(* POU HTML_DECODE, ST *)
FUNCTION HTML_DECODE : STRING(255)
VAR_INPUT
	IN : STRING(255);
END_VAR
VAR
	pos : INT;
	end : INT;
	tmp : STRING(10);
	code : STRING(1);
END_VAR


(*
version 1.2		17. dec. 2008
programmer 		hugo
tested by		oscat

HTML_DECODE converts HTML coded characters to text. 
&amp; is replaced by & ("Ampersand")
&lt; is replaced by < ("lower than")
&gt; is replaced by > ("greater than")
&quot; is replaced by " ("Quote")
all other &names characters are replaced by their respective character codes.

*)
HTML_DECODE := IN;

(* docode characters encoded by character position *)
pos := FIND(HTML_DECODE, '&');
WHILE pos > 0 DO
	tmp := MID(HTML_DECODE, 2, pos + 1);
	IF tmp = '#x' OR tmp = '#X' THEN
		(* hexadecimal representation found *)
		tmp := MID(HTML_DECODE, 10, pos + 3);
		end := FIND(tmp, ';');
		CODE := CHR_TO_STRING(DWORD_TO_BYTE(HEX_TO_DWORD(LEFT(tmp, end - 1))));
		HTML_DECODE := REPLACE(HTML_DECODE, CODE, end + 3, pos);
	ELSIF LEFT(tmp,1) = '#' THEN
		tmp := MID(HTML_DECODE, 10, pos + 2);
		end := FIND(tmp, ';');
		CODE := CHR_TO_STRING(INT_TO_BYTE(STRING_TO_INT(LEFT(tmp, end - 1))));
		HTML_DECODE := REPLACE(HTML_DECODE, CODE, end + 2, pos);
	ELSE
		(* replace all named characters *)
		tmp := MID(HTML_DECODE, 10, pos + 1);
		end := FIND(tmp, ';');
		CODE := CHR_TO_STRING(CHARCODE(LEFT(tmp, end - 1)));
		HTML_DECODE := REPLACE(HTML_DECODE, CODE, end + 1, pos);
	END_IF;
	(* search for next occurence of encoded characters *)
	pos := FINDP(HTML_DECODE, '&', pos + 1);
END_WHILE;



(* revision history
hm	3. mai. 2008	rev 1.0
	original version

hm	16. jun. 2008	rev 1.1
	changed nested call of replace for better compatibility

hm	17. dec. 2008	rev 1.2
	changed function CHR to CHR_TO_STRING

*)
END_FUNCTION

(* POU HTML_ENCODE, ST *)
FUNCTION HTML_ENCODE : STRING(255)
VAR_INPUT
	IN : STRING(255);
	M : BOOL;
END_VAR
VAR
	pt_in : POINTER TO ARRAY[1..255] OF BYTE;
	pt_out : POINTER TO ARRAY[1..256] OF BYTE;
	pos_in : INT;
	pos_out : INT;
	stop : INT;
	B: BYTE;
	tmp : STRING(10);
	i: INT;
END_VAR


(*
version 1.0		3. mai. 2008
programmer 		hugo
tested by		hugo 

HTML_ENCODE checks a string if it contains reserved HTML characters and converts them to alternative html coding.
& is replaced by &amp; ("Ampersand")
< is replaced by &lt; ("lower than")
> is replaced by &gt; ("greater than")
" is replaced by &quot; ("Quote")

*)
pt_in  := ADR(in);
pt_out := ADR(HTML_ENCODE);

(* scan the input string and convert unallowed characters *)
pos_in := 1;
stop := LEN(in);
FOR pos_out := 1 TO 255 DO
	IF pos_in > stop THEN EXIT; END_IF;
	B := pt_in^[pos_in];
	CASE BYTE_TO_INT(B) OF
		34: (* " detected *)
			IF pos_out > 249 THEN EXIT; END_IF;
			pt_out^[pos_out] := 38;
			pos_out := pos_out + 1;
			pt_out^[pos_out] := 113;
			pos_out := pos_out + 1;
			pt_out^[pos_out] := 117;
			pos_out := pos_out + 1;
			pt_out^[pos_out] := 111;
			pos_out := pos_out + 1;
			pt_out^[pos_out] := 116;
			pos_out := pos_out + 1;
			pt_out^[pos_out] := 59;
		38: (* & detected *)
			IF pos_out > 250 THEN EXIT; END_IF;
			pt_out^[pos_out] := 38;
			pos_out := pos_out + 1;
			pt_out^[pos_out] := 97;
			pos_out := pos_out + 1;
			pt_out^[pos_out] := 109;
			pos_out := pos_out + 1;
			pt_out^[pos_out] := 112;
			pos_out := pos_out + 1;
			pt_out^[pos_out] := 59;
		60: (* < detected *)
			IF pos_out > 251 THEN EXIT; END_IF;
			pt_out^[pos_out] := 38;
			pos_out := pos_out + 1;
			pt_out^[pos_out] := 108;
			pos_out := pos_out + 1;
			pt_out^[pos_out] := 116;
			pos_out := pos_out + 1;
			pt_out^[pos_out] := 59;
		62: (* > detected *)
			IF pos_out > 251 THEN EXIT; END_IF;
			pt_out^[pos_out] := 38;
			pos_out := pos_out + 1;
			pt_out^[pos_out] := 103;
			pos_out := pos_out + 1;
			pt_out^[pos_out] := 116;
			pos_out := pos_out + 1;
			pt_out^[pos_out] := 59;
	ELSE
		IF M AND B > 127 THEN
			tmp := CHARNAME(B);
			(* exit if output string has not enough space *)
			IF pos_out + LEN(tmp) + 2 <= 255 THEN
				pt_out^[pos_out] := 38;
				pos_out := pos_out + 1;
				FOR i := 1 TO LEN(tmp) DO
					pt_out^[pos_out] := CODE(tmp, i);
					pos_out := pos_out + 1;
				END_FOR;
				pt_out^[pos_out] := 59;
			END_IF;
		ELSE
			pt_out^[pos_out] := B;
		END_IF;
	END_CASE
	(* increment in by 1 *)
	pos_in := pos_in + 1;
END_FOR;

(* terminate the output string *)
pt_out^[pos_out] := 0;



(* revision history
hm		3. mai. 2008	rev 1.0
	original version

*)
END_FUNCTION

(* POU HYST, ST *)
FUNCTION_BLOCK HYST
VAR_INPUT
	In : REAL;
	ON : REAL;
	OFF : REAL;
END_VAR
VAR_OUTPUT
	Q : BOOL;
	win : BOOL;
END_VAR
VAR
END_VAR

(*
version 1.0	2. jun. 2008
programmer 	hugo
tested BY	oscat

This Hystereses function has two modes:
1. if on > off then Q will be switched high when in > on and switched low when in < off.
2. if on < off then Q will be switched high when in < on and switched low when in > off.
the output win will be high when in is between low and high.

*)
IF ON >= OFF THEN
	IF IN < OFF THEN
		Q := FALSE;
		WIN := FALSE;
	ELSIF  IN > ON THEN
		Q := TRUE;
		WIN := FALSE;
	ELSE
		WIN := TRUE;
	END_IF;
ELSE
	IF IN > OFF THEN
		Q := FALSE;
		WIN := FALSE;
	ELSIF  IN < ON THEN
		Q := TRUE;
		WIN := FALSE;
	ELSE
		WIN := TRUE;
	END_IF;
END_IF;


(* revision history
hm		2.  jun 2008	rev 1.0
	original version

*)
END_FUNCTION_BLOCK

(* POU HYST_1, ST *)
FUNCTION_BLOCK HYST_1
VAR_INPUT
	In : REAL;
	high : REAL;
	low : REAL;
END_VAR
VAR_OUTPUT
	Q : BOOL;
	win : BOOL;
END_VAR
VAR
END_VAR

(*
version 1.1	2. jun. 2008
programmer 	hugo
tested BY	oscat

this hysteresis function switches the output high if the input signal reaches obove high and will switch to low when the input falls back below low value.
a separate output mid is set if the input stays between low and high value.

*)
IF in < low THEN
	Q := FALSE;
	win := FALSE;
ELSIF in > high THEN
	Q := TRUE;
	win := FALSE;
ELSE
	win := TRUE;
END_IF;

(* code used for rev 1.0
IF Q THEN
	IF in < low THEN q := FALSE; END_IF;
ELSE
	IF in > high THEN q := TRUE; END_IF;
END_IF;
win := in > low AND in < high;
*)


(* revision history
hm		4.  aug. 2006	rev 1.0
	original version

hm		2. jun. 2008	rev 1.1
	improved performance
*)
END_FUNCTION_BLOCK

(* POU HYST_2, ST *)
FUNCTION_BLOCK HYST_2
VAR_INPUT
	IN : REAL;
	VAL : REAL;
	HYS : REAL;
END_VAR
VAR_OUTPUT
	Q : BOOL;
	WIN: BOOL;
END_VAR
VAR
	tmp: REAL;
END_VAR


(*
version 1.2	2. jun. 2008
programmer 	oscat
tested BY	oscat

this hysteresis function switches the output high if the input signal reaches obove val + hys/2 and will switch to low when the input falls back below val - hys/2 value.
a separate output mid is set if the input stays between low and high value.

*)
tmp := val - hys * 0.5;
IF in < tmp THEN
	Q := FALSE;
	win := FALSE;
ELSIF in > tmp + hys THEN
	Q := TRUE;
	win := FALSE;
ELSE
	win := TRUE;
END_IF;

(* code used for 1.2 and before
X := hys * 0.5;
IF Q THEN
	IF in < val - x THEN q := FALSE; END_IF;
ELSE
	IF in > val + x THEN q := TRUE; END_IF;
END_IF;
win := in > val - x AND in < val + x;
*)

(* revision history
hm		4. aug 2006	rev 1.0
	original version

hm		5. jan 2008	rev 1.1
	improved code for better performance

hm		2. jun. 2008	rev 1.2
	improved performance
*)
END_FUNCTION_BLOCK

(* POU HYST_3, ST *)
FUNCTION_BLOCK HYST_3
VAR_INPUT
	in : REAL;
	hyst : REAL;
	val1 : REAL;
	val2 : REAL;
END_VAR
VAR_OUTPUT
	Q1 : BOOL;
	Q2 : BOOL;
END_VAR
VAR
	X: REAL;
END_VAR

(*
version 1.2	5 jan 2008
programmer 	oscat
tested BY	oscat

this is a double hysteresis function. Out1 follows a hysteresis function defined by val1and hyst, while out 2 follows val2 and hyst.
if the input signal is between the two hysteresis switches (val1 and val2) then non of the outputs is active.

*)
X := hyst * 0.5;
IF in < val1 - X THEN
	q1 := TRUE;
ELSIF in > val1 + X THEN
	q1 := FALSE;
END_IF;
IF in < val2 - X THEN
	q2 := FALSE;
ELSIF in > val2 + X THEN
	q2 := TRUE;
END_IF;

(* revision history
hm	22. jan 2007	rev 1.0
	original version

hm	27. dec 2007	rev 1.1
	changed code for better performance

hm	5. jan 2008	rev 1.2
	further performance iprovements

*)
END_FUNCTION_BLOCK

(* POU INC_DEC, ST *)
FUNCTION_BLOCK INC_DEC
VAR_INPUT
	CHa : BOOL;
	CHb : BOOL;
	RST : BOOL;
END_VAR
VAR_OUTPUT
	dir : BOOL;
	cnt : INT;
END_VAR
VAR
	edgea : BOOL;
	clk: BOOL;
	clka: BOOL;
	clkb: BOOL;
	edgeb: BOOL;
	axb: BOOL;
END_VAR

(*
	version 1.0	4 aug 2006
	programmer 	oscat
	tested BY		oscat

incremental decoder with quadruple accuracy.
2 pulses for each channel are created for each directional pulse.
*)
axb := cha XOR chb;

(* create pulses for channel a *)
clka := cha XOR edgea;
edgea := cha;

clkb := chb XOR edgeb;
edgeb := chb;

(* create pulses for both channels *)
clk := clka OR clkb;

(* set the direction output *)
IF axb AND clka THEN dir := TRUE; END_IF;
IF axb AND clkb THEN dir := FALSE; END_IF;

(* increment or decrement the counter *)
IF clk AND dir THEN cnt := cnt + 1; END_IF;
IF clk AND NOT dir THEN cnt := cnt -1; END_IF;

(* reset the counter if rst active *)
IF rst THEN cnt := 0; END_IF;
END_FUNCTION_BLOCK

(* POU INT_TO_BCDC, ST *)
FUNCTION INT_TO_BCDC : BYTE
VAR_INPUT
	IN : INT;
END_VAR
VAR
END_VAR

(*
version 1.1	30. jun. 2008
programmer 	hugo
tested by		tobias

this function converts an integer into a two digit bcd number.
*)
INT_TO_BCDC := SHL(INT_TO_BYTE(IN / INT#10),4) OR INT_TO_BYTE(in MOD INT#10);

(* revision history
hm	13.12.2007
	original version

hm	30.6.2008	rev 1.1
	changed name INT_TO_BCD to INT_TO_BCDC to avoid collision with util.lib
	corrected error in code

*)
END_FUNCTION

(* POU INTERLOCK_4, ST *)
FUNCTION_BLOCK INTERLOCK_4
VAR_INPUT CONSTANT
END_VAR
VAR_INPUT
	I0 : BOOL;
	I1 : BOOL;
	I2 : BOOL;
	I3 : BOOL;
	E : BOOL;
	MODE : INT;

END_VAR
VAR_OUTPUT
	OUT : BYTE;
	TP : BOOL;
END_VAR
VAR
	in: BYTE;
	last: BYTE;
	old: BYTE;
	lmode: INT;
END_VAR

(*
version 1.0	24. oct. 2008
programmer 	hugo
tested by	oscat

INTERLOCK_4 detects one of 4 switches and delivers the number of the switch pressed on the output out
a output tp is true for one cycle if the output has changed.
a setup variable MODE selects between 3 different modes:
MODE = 0, any input active will disable all other inputs
MODE = 1, the input with the highest number will be acepted
mode = 2, the input last pressed will disable all others 

*)
(* check if enable is active *)
IF E THEN
(* reset all vars when there is a mode change on thy fly *)
	IF mode <> lmode THEN
		out := last := old := 0;
		lmode := mode;
	END_IF;
	(* load inputs into in *)
	in.0 := I0;	in.1 := I1;	in.2 := I2;	in.3 := I3;
	(* only execute when there is any change *)
	IF in <> last THEN
		(* only execute when inputs have chages state *)
		CASE mode OF
			0:	(* output directly display inputs as bits in byte out *)
				out := in;

			1:	(* the input with the highest number will be acepted *)
				IF in.3 THEN out := 8;
				ELSIF in.2 THEN out := 4;
				ELSIF in.1 THEN out := 2;
				ELSE out := in;
				END_IF;

			2:	(* input last pressed will be displayed only *)
				last := ((in XOR last) AND in);
				IF last.3 THEN out := 8;
				ELSIF last.2 THEN out := 4;
				ELSIF last.1 THEN out := 2;
				ELSE out := last;
				END_IF;

			3:	(* any input active will disable all other inputs *)
				IF (out AND in) = 0 THEN
					IF in.3 THEN out := 8;
					ELSIF in.2 THEN out := 4;
					ELSIF in.1 THEN out := 2;
					ELSE out := in;
					END_IF;
				END_IF;

		END_CASE;
		last := in;
	END_IF;
	tp := out <> old;
	old := out;
ELSE
	out := last := old := 0;
	lmode := 0;
	tp := FALSE;
END_IF;





(* revision history
hm	24. oct 2008	rev 1.0
	original version

*)
END_FUNCTION_BLOCK

(* POU IP4_CHECK, ST *)
FUNCTION IP4_CHECK : BOOL
VAR_INPUT
	NIP : DWORD;
	LIP : DWORD;
	SM : DWORD;
END_VAR
VAR
END_VAR

(*
version 1.0	4. mar 2008
programmer 	hugo
tested by		oscat

IP4_CHECK testet ob eine Network IP und Local_IP im selben Subnet sind.

*)
IP4_CHECK := (NIP AND sm) = (LIP AND SM);


(* revision history
hm		4. mar 2008	rev 1.0
	original version

*)
END_FUNCTION

(* POU IP4_DECODE, ST *)
FUNCTION IP4_DECODE : DWORD
VAR_INPUT
	str : STRING;
END_VAR
VAR
	d1, d2, d3, d4 : INT;
	s1, s2, s3, s4 : STRING(3);
END_VAR

(*
version 1.0	29. feb 2008
programmer 		kurt
tested by		hugo

IP4_DECODE testet ob ein string eine gültige IPv4 Adresse enthält und gibt die 4 Bytes der IP Adresse als DWORD zurück.

*)
IP4_DECODE := 0;
(* check wheather 3 dots are present *)
IF COUNT_CHAR(str,46) <> 3 THEN RETURN; END_IF;
(* store the positions of the 3 dots *)
d1 := FINDP(str,'.',1);
d2 := FINDP(str,'.',d1+1);
d3 := FINDP(str,'.',d2+1);
IF d1 > 4 OR d2 - d1 > 4 OR d3 - d2 > 4 THEN RETURN; END_IF;
(* store the 3 strings between the dots in d1 .. d4 *)
s1 := LEFT(str,d1-1);
s2 := MID(str,d2-d1-1,d1+1);
s3 := MID(str,d3-d2-1,d2+1);
s4 := RIGHT(str,LEN(str)-d3);
(* check if the 3 strings are numbers only *)
IF NOT IS_NUM(s1) OR NOT IS_NUM(s2) OR NOT IS_NUM(s3) OR NOT IS_NUM(s4) THEN RETURN; END_IF;
(* convert the 4 numbers and check range 0..255 *)
d1 := STRING_TO_INT(s1);
d2 := STRING_TO_INT(s2);
d3 := STRING_TO_INT(s3);
d4 := STRING_TO_INT(s4);
(* check range of numbers *)
IF d1 > 255 OR d2 > 255 OR d3 > 255 OR d4 > 255 THEN RETURN; END_IF;
(* convert to output *)
IP4_DECODE := SHL(INT_TO_DWORD(d1),24) OR SHL(INT_TO_DWORD(d2),16) OR SHL(INT_TO_DWORD(d3),8) OR INT_TO_DWORD(d4);



(* revision history
hm		29. feb 2008	rev 1.0
	original version

*)
END_FUNCTION

(* POU IS_NUM, ST *)
FUNCTION IS_NUM : BOOL
VAR_INPUT
	str : STRING(STRING_LENGTH);
END_VAR
VAR
	L : INT;
	pt : POINTER TO BYTE;
	pos: INT;
END_VAR

(*
version 1.1	29. mar. 2008
programmer 		kurt
tested by		hugo

IS_NUM testet ob in einem string nur Zahlen 0..9 vorkommen.

*)
PT := ADR(str);
L := LEN(str);
FOR pos := 1 TO L DO
	IF NOT (ISC_NUM(pt^)) THEN
		IS_NUM := FALSE;
		RETURN;
	END_IF;
    	PT := PT + 1;
END_FOR;
IS_NUM := L > 0;


(* revision history
hm	29. feb 2008	rev 1.0
	original version

hm	29. mar. 2008	rev 1.1
	changed STRING to STRING(STRING_LENGTH)
*)
END_FUNCTION

(* POU ISC_NUM, ST *)
FUNCTION ISC_NUM : BOOL
VAR_INPUT
	IN : BYTE;
END_VAR
VAR
END_VAR

(*
version 1.0	6. mar 2008
programmer 	oscat
tested by		hugo

ISC_NUM checks if a character is 0..9.

*)
ISC_NUM := IN > 47 AND IN < 58;

(* revision history
hm		6. mar. 2008	rev 1.0
	original version

*)
END_FUNCTION

(* POU IP4_TO_STRING, ST *)
FUNCTION IP4_TO_STRING : STRING(15)
VAR_INPUT
	IP4 : DWORD;
END_VAR
VAR
	tmp : STRING(3);
END_VAR

(*
version 1.0	22. apr. 2008
programmer 	kurt
tested by		hugo

IP4_TO_STRING erzeugt eine IP Adresse als String aus einem DWORD..

*)
IP4_TO_STRING := DWORD_TO_STRING(SHR(IP4, 24));
IP4_TO_STRING := CONCAT(IP4_TO_STRING, '.');
tmp := DWORD_TO_STRING(SHR(SHL(ip4,8), 24));
IP4_TO_STRING := CONCAT(IP4_TO_STRING, tmp);
IP4_TO_STRING := CONCAT(IP4_TO_STRING, '.');
tmp := DWORD_TO_STRING(SHR(SHL(ip4,16), 24));
IP4_TO_STRING := CONCAT(IP4_TO_STRING, tmp);
IP4_TO_STRING := CONCAT(IP4_TO_STRING, '.');
tmp := DWORD_TO_STRING(SHR(SHL(ip4, 24), 24));
IP4_TO_STRING := CONCAT(IP4_TO_STRING, tmp);


(* revision history
hm		22. apr 2008	rev 1.0
	original version

*)
END_FUNCTION

(* POU IRTRANS_1, ST *)
FUNCTION_BLOCK IRTRANS_1
VAR_INPUT CONSTANT
	DEV_CODE : STRING;
	KEY_CODE : STRING;
END_VAR
VAR_INPUT
	CMD : BOOL;
END_VAR
VAR_IN_OUT
	DEV : STRING;
	KEY : STRING;
END_VAR
VAR_OUTPUT
	Q : BOOL;
END_VAR
VAR
END_VAR

(*
version 1.2	19. oct. 2008
programmer 	hugo
tested BY	oscat

*)
Q := cmd AND dev_code = dev AND key_code = key;

(* revision history
hm	2. jan 2008		rev 1.0
	original version

hm	20. 6. 2008		rev 1.1
	performance improvement

hm	19. oct. 2008	rev 1.2
	changed input device_code to dev_code and device to dev for compatibility reasons

*)
END_FUNCTION_BLOCK

(* POU IRTRANS_4, ST *)
FUNCTION_BLOCK IRTRANS_4
VAR_INPUT CONSTANT
	DEV_CODE : STRING;
	KEY_CODE_0 : STRING;
	KEY_CODE_1 : STRING;
	KEY_CODE_2 : STRING;
	KEY_CODE_3 : STRING;
END_VAR
VAR_INPUT
	CMD : BOOL;
END_VAR
VAR_IN_OUT
	DEV : STRING;
	KEY : STRING;
END_VAR
VAR_OUTPUT
	Q0, Q1, Q2, Q3 : BOOL;
END_VAR
VAR_TEMP
	decode: BOOL;
END_VAR

(*
version 1.2	19. oct. 2008
programmer 	hugo
tested BY	oscat

*)
decode := cmd AND dev_code = dev;

Q0 := key = key_code_0 AND decode;
Q1 := key = key_code_1 AND decode;
Q2 := key = key_code_2 AND decode;
Q3 := key = key_code_3 AND decode;



(* revision history
hm	2. jan 2008		rev 1.0
	original version

hm	17. oct. 2008	rev 1.1
	improved performance

hm	19. oct. 2008	rev 1.2
	changed input device_code to dev_code and device to dev for compatibility reasons
*)
END_FUNCTION_BLOCK

(* POU IRTRANS_8, ST *)
FUNCTION_BLOCK IRTRANS_8
VAR_INPUT CONSTANT
	dev_code : STRING;
	key_code_0 : STRING;
	key_code_1 : STRING;
	key_code_2 : STRING;
	key_code_3 : STRING;
	key_code_4 : STRING;
	key_code_5 : STRING;
	key_code_6 : STRING;
	key_code_7 : STRING;
END_VAR
VAR_INPUT
	CMD : BOOL;
END_VAR
VAR_IN_OUT
	DEV : STRING;
	KEY : STRING;
END_VAR
VAR_OUTPUT
	Q0, Q1, Q2, Q3, Q4, Q5, Q6, Q7 : BOOL;
END_VAR
VAR_TEMP
	decode: BOOL;
END_VAR

(*
version 1.2	19. oct. 2008
programmer 	hugo
tested BY	oscat

*)
decode := cmd AND dev_code = dev;

Q0 := key = key_code_0 AND decode;
Q1 := key = key_code_1 AND decode;
Q2 := key = key_code_2 AND decode;
Q3 := key = key_code_3 AND decode;
Q4 := key = key_code_4 AND decode;
Q5 := key = key_code_5 AND decode;
Q6 := key = key_code_6 AND decode;
Q7 := key = key_code_7 AND decode;


(* revision history
hm	2. jan 2008		rev 1.0
	original version

hm	17. oct 2008	rev 1.1
	improved performance

hm	19. oct. 2008	rev 1.2
	changed input device_code to dev_code and device to dev for compatibility reasons

*)
END_FUNCTION_BLOCK

(* POU IRTRANS_DECODE, ST *)
FUNCTION_BLOCK IRTRANS_DECODE
VAR_INPUT
	BUFFER : POINTER TO ARRAY[0..32000] OF BYTE;
END_VAR
VAR_IN_OUT
	LENGTH : DINT;
END_VAR
VAR_OUTPUT
	CMD : BOOL;
	DEV : STRING;
	KEY : STRING;
	ERROR : BOOL;
END_VAR
VAR
	pt : POINTER TO BYTE;
	i : INT;
	stop : INT;
END_VAR

(*
version 1.1	19. oct. 2008
programmer 	hugo
tested BY	tobias

*)
(* do nothing if the buffer is empty *)
IF DINT_TO_INT(length) > 0 THEN
	i := 0;
	error := TRUE;
	stop := DINT_TO_INT(length) - 2;
	(* read characters before first comma and store in device *)
	pt := ADR(dev);
	WHILE i < stop DO
		IF buffer^[i] = 44 THEN EXIT; END_IF;
		pt^ := buffer^[i];
		pt := pt + 1;
		i := i + 1;
	END_WHILE;
	(* terminate the device string *)
	pt^ := 0;
	(* read after first comma and store in key *)
	i := i + 1;
	pt := ADR(key);
	WHILE i < stop DO
		pt^ := buffer^[i];
		pt := pt + 1;
		i := i + 1;
	END_WHILE;
	(* terminate the key string *)
	pt^:= 0;
	(* check if last two characters are $R$N 13, 10 *)
	IF buffer^[i] <> 13 AND buffer^[i+1] <> 10 THEN	RETURN;	END_IF;
	(* check if device and key are present *)
	IF LEN(dev) = 0 OR LEN(key) = 0 THEN RETURN; END_IF;
	(* a valid transmission has been received *)
	cmd := TRUE;
	error := FALSE;
	(* clear the input buffer to allow the next transmission to occur *)
	length := 0;
ELSE
	error := cmd := FALSE;
END_IF;


(* revision history
hm	2. jan 2008		rev 1.0
	original version

hm	19. oct. 2008	rev 1.1
	added typecast to avoid warnings
	changed output device to dev for compatibility reasons

*)
END_FUNCTION_BLOCK

(* POU IS_ALNUM, ST *)
FUNCTION IS_ALNUM : BOOL
VAR_INPUT
	str : STRING(STRING_LENGTH);
END_VAR
VAR
	L: INT;
	pt : POINTER TO BYTE;
	pos: INT;
END_VAR

(*
version 1.1	29. mar. 2008
programmer 		kurt
tested by		hugo

ISC_ALNUM testet ob in einem string nur Zahlen 0..9 vorkommen.

*)
PT := ADR(str);
L := LEN(str);
FOR pos := 1 TO L DO
	IF NOT (ISC_ALPHA(pt^) OR ISC_NUM(pt^)) THEN
		IS_ALNUM := FALSE;
		RETURN;
	END_IF;
    	PT := PT + 1;
END_FOR;
IS_ALNUM := L > 0;


(* revision history
hm	29. feb 2008	rev 1.0
	original version

hm	29. mar. 2008	rev 1.1
	changed STRING to STRING(STRING_LENGTH)
*)
END_FUNCTION

(* POU ISC_ALPHA, ST *)
FUNCTION ISC_ALPHA : BOOL
VAR_INPUT
	IN : BYTE;
END_VAR
VAR
END_VAR

(*
version 1.1	19. oct. 2008
programmer 	oscat
tested by	oscat

ISC_ALPHA checks if a character is a..z or A..Z.

*)
IF setup.EXTENDED_ASCII THEN
	ISC_ALPHA := (in > 64 AND in < 91) OR (in > 191  AND in <> 215 AND in <> 247) OR (in > 96 AND in < 123);
ELSE
	ISC_ALPHA := (IN > 64 AND IN < 91) OR (in > 96 AND in < 123);
END_IF;

(* revision history
hm	6. mar. 2008	rev 1.0
	original version

hm	19. oct. 2008	rev 1.1
	changes setup constants
*)
END_FUNCTION

(* POU IS_ALPHA, ST *)
FUNCTION IS_ALPHA : BOOL
VAR_INPUT
	str : STRING(STRING_LENGTH);
END_VAR
VAR
	L: INT;
	pt : POINTER TO BYTE;
	pos: INT;
END_VAR

(*
version 1.1	29. mar. 2008
programmer 		kurt
tested by		hugo

IS_ALPHA testet ob in einem string nur Zeichen a-z oder A - Z vorkommen.

*)
PT := ADR(str);
L := LEN(str);
FOR pos := 1 TO L DO
	IF NOT ISC_ALPHA(pt^) THEN
		IS_ALPHA := FALSE;
		RETURN;
	END_IF;
    	PT := PT + 1;
END_FOR;
IS_ALPHA := L > 0;


(* revision history
hm	29. feb 2008	rev 1.0
	original version

hm	29. mar. 2008	rev 1.1
	changed STRING to STRING(STRING_LENGTH)
*)
END_FUNCTION

(* POU IS_CC, ST *)
FUNCTION IS_CC : BOOL
VAR_INPUT
	str : STRING(STRING_LENGTH);
	cmp : STRING(STRING_LENGTH);
END_VAR
VAR
	L: INT;
	pos: INT;
END_VAR

(*
version 1.1	29. mar. 2008
programmer 	Tobias
tested by	hugo

ISC_CC testet ob ein string nur aus Zeichen des Strings CMP besteht.

*)
L := LEN(str);
FOR pos := 1 TO L DO
	IF FIND(CMP,MID(str,1,pos)) = 0 THEN RETURN; END_IF;
END_FOR;
IS_CC := L > 0;



(* revision history
hm	19. mar 2008	rev 1.0
	original version

hm	29. mar. 2008	rev 1.1
	changed STRING to STRING(STRING_LENGTH)
*)
END_FUNCTION

(* POU IS_CTRL, ST *)
FUNCTION IS_CTRL : BOOL
VAR_INPUT
	str : STRING(STRING_LENGTH);
END_VAR
VAR
	L: INT;
	pt : POINTER TO BYTE;
	pos: INT;
END_VAR

(*
version 1.1	29. mar 2008
programmer 		kurt
tested by		hugo

IS_CTRL testet ob in einem string nur Steuerzeichen (Char < 32) vorkommen.

*)
PT := ADR(str);
L := LEN(str);
FOR pos := 1 TO L DO
	IF NOT (ISC_CTRL(pt^)) THEN
		IS_CTRL := FALSE;
		RETURN;
	END_IF;
    	PT := PT + 1;
END_FOR;
IS_CTRL := L > 0;


(* revision history
hm	29. feb. 2008	rev 1.0
	original version

hm	29. mar. 2008	rev 1.1
	changed STRING to STRING(STRING_LENGTH)
*)
END_FUNCTION

(* POU ISC_CTRL, ST *)
FUNCTION ISC_CTRL : BOOL
VAR_INPUT
	IN : BYTE;
END_VAR
VAR
END_VAR

(*
version 1.0	6. mar 2008
programmer 	oscat
tested by		hugo

ISC_ALPHA checks if a character is a control character.

*)
ISC_CTRL := IN < 32 OR IN = 127;

(* revision history
hm		6. mar. 2008	rev 1.0
	original version

*)
END_FUNCTION

(* POU IS_HEX, ST *)
FUNCTION IS_HEX : BOOL
VAR_INPUT
	str : STRING(STRING_LENGTH);
END_VAR
VAR
	L: INT;
	pt : POINTER TO BYTE;
	pos: INT;
END_VAR

(*
version 1.1	29. mar. 2008
programmer 		kurt
tested by		hugo

IS_HEX testet ob in einem string nur Zahlen 0..9 oder A..F oder a..f  vorkommen.

*)
PT := ADR(str);
L := LEN(str);
FOR pos := 1 TO L DO
	IF NOT (ISC_HEX(pt^)) THEN
		IS_HEX := FALSE;
		RETURN;
	END_IF;
    	PT := PT + 1;
END_FOR;
IS_HEX := L > 0;


(* revision history
hm	29. feb 2008	rev 1.0
	original version

hm	29. mar. 2008	rev 1.1
	changed STRING to STRING(STRING_LENGTH)
*)
END_FUNCTION

(* POU ISC_HEX, ST *)
FUNCTION ISC_HEX : BOOL
VAR_INPUT
	IN : BYTE;
END_VAR
VAR
END_VAR

(*
version 1.0	6. mar 2008
programmer 	oscat
tested by		hugo

ISC_HEX checks if a character is 0..9, A..F, a..f.

*)
ISC_HEX := (IN > 47 AND IN < 58) OR (IN > 64 AND IN < 71) OR (IN > 96 AND IN < 103);

(* revision history
hm		6. mar. 2008	rev 1.0
	original version

*)
END_FUNCTION

(* POU IS_IP4, ST *)
FUNCTION IS_IP4 : BOOL
VAR_INPUT
	str : STRING;
END_VAR
VAR
END_VAR

(*
version 1.0	1. mar 2008
programmer 		kurt
tested by		hugo

IS_IP4 testet ob ein string eine gültige IPv4 Adresse enthält.

*)
IS_IP4 := IP4_DECODE(str) > 0;


(* revision history
hm		1. mar 2008	rev 1.0
	original version

*)
END_FUNCTION

(* POU IS_LOWER, ST *)
FUNCTION IS_LOWER : BOOL
VAR_INPUT
	str : STRING(STRING_LENGTH);
END_VAR
VAR
	l: INT;
	pt : POINTER TO BYTE;
	pos: INT;
END_VAR

(*
version 1.1	29. mar. 2008
programmer 		kurt
tested by		hugo

IS_LOWER testet ob in einem string nur kleinbuchstaben vorkommen.

*)
PT := ADR(str);
L := LEN(str);
FOR pos := 1 TO L DO
	IF NOT (ISC_LOWER(pt^)) THEN
		IS_LOWER := FALSE;
		RETURN;
	END_IF;
    	PT := PT + 1;
END_FOR;
IS_LOWER := L > 0;


(* revision history
hm	29. feb 2008	rev 1.0
	original version

hm	29. mar. 2008	rev 1.1
	changed STRING to STRING(STRING_LENGTH)
*)
END_FUNCTION

(* POU ISC_LOWER, ST *)
FUNCTION ISC_LOWER : BOOL
VAR_INPUT
	IN : BYTE;
END_VAR
VAR
END_VAR

(*
version 1.1	19. oct. 2008
programmer 	hugo
tested by	oscat

isc_lower checks if a character is lowercase.

*)
IF setup.EXTENDED_ASCII THEN
	ISC_LOWER := ((in > 96) AND (in < 123)) OR ((in > 222) AND (in <> 247));
ELSE
	ISC_LOWER := ((in > 96) AND (in < 123));
END_IF;

(* revision history
hm	6. mar. 2008	rev 1.0
	original version

hm	19. oct. 2008	rev 1.1
	changes setup constants
*)
END_FUNCTION

(* POU IS_NCC, ST *)
FUNCTION IS_NCC : BOOL
VAR_INPUT
	str : STRING(STRING_LENGTH);
	cmp : STRING(STRING_LENGTH);
END_VAR
VAR
	L: INT;
	pos: INT;
END_VAR

(*
version 1.1	29. mar. 2008
programmer 		Tobias
tested by		hugo

ISC_NCC testet ob in einem string keine Zeichen des Strings CMP enthalten sind.

*)
L := LEN(str);
FOR pos := 1 TO L DO
	IF FIND(CMP,MID(str,1,pos)) > 0 THEN RETURN; END_IF
END_FOR;
IS_NCC := TRUE;



(* revision history
hm	19. mar 2008	rev 1.0
	original version

hm	29. mar. 2008	rev 1.1
	changed STRING to STRING(STRING_LENGTH)
*)
END_FUNCTION

(* POU IS_SORTED, ST *)
FUNCTION IS_SORTED : BOOL
VAR_INPUT
	pt : POINTER TO ARRAY[0..32000] OF REAL;
	size : UINT;
END_VAR
VAR

	stop: INT;
	i: INT;
END_VAR

(*
version 1.1	4. apr. 2008
programmer 	hugo
tested by	tobias

this function will return true if the given array is sorted in an ascending order.
the function needs to be called:	array_sorted(adr("array"),sizeof("array"));
because this function works with pointers its very time efficient and it needs no extra memory.

*)
stop := UINT_TO_INT(SHR(size,2)-2);
FOR i := 0 TO stop DO
	IF pt^[i] > pt^[i+1] THEN
		IS_SORTED := FALSE;
		RETURN;
	END_IF;
END_FOR;

IS_SORTED := TRUE;

(* revision history

hm 	29. mar. 2008 	rev 1.0
	original version

hm	4. apr. 2008	rev 1.1
	added type conversion to avoid warnings under codesys 3.0
*)
END_FUNCTION

(* POU IS_UPPER, ST *)
FUNCTION IS_UPPER : BOOL
VAR_INPUT
	str : STRING(STRING_LENGTH);
END_VAR
VAR
	L: INT;
	pt : POINTER TO BYTE;
	pos: INT;
END_VAR

(*
version 1.1	29. mar. 2008
programmer 		kurt
tested by		hugo

IS_UPPER testet ob in einem string keine Kleinbuchstaben vorkommen.

*)
PT := ADR(str);
L := LEN(str);
FOR pos := 1 TO L DO
	IF NOT (ISC_UPPER(pt^)) THEN
		IS_UPPER := FALSE;
		RETURN;
	END_IF;
    	PT := PT + 1;
END_FOR;
IS_UPPER := L > 0;


(* revision history
hm	29. feb 2008	rev 1.0
	original version

hm	29. mar. 2008	rev 1.1
	changed STRING to STRING(STRING_LENGTH)
*)
END_FUNCTION

(* POU ISC_UPPER, ST *)
FUNCTION ISC_UPPER : BOOL
VAR_INPUT
	IN : BYTE;
END_VAR
VAR
END_VAR

(*
version 1.1	19. oct. 2008
programmer 	hugo
tested by	oscat

ISC_upper checks if a character is uppercase

*)
IF setup.EXTENDED_ASCII THEN
	ISC_UPPER :=  ((in > 64) AND (in < 91)) OR (((in > 191) AND (in < 223)) AND (in <> 215));
ELSE
	ISC_UPPER := ((in > 64) AND (in < 91));
END_IF;


(* revision history
hm	6. mar. 2008	rev 1.0
	original version

hm	19. oct. 2008	rev 1.1
	changes setup constants

*)
END_FUNCTION

(* POU IS_URLCHR, ST *)
FUNCTION IS_URLCHR : BOOL
VAR_INPUT
	IN : BYTE;
END_VAR
VAR
END_VAR

(*
version 1.0		27. apr. 2008
programmer 		hugo
tested by		hugo

IS_URL_CHR is true if a string contains only non reserved characters for an url.
the non reserved characters are : [A..Z], [a..z], [0..9], -_.~

*)
IS_URLCHR := ((IN > 47) AND (IN < 58)) OR ((IN > 64) AND (IN < 91)) OR ((IN > 96) AND (IN < 123)) OR (in = 126) OR (in = 95) OR (in =45) OR (in =46);


(* revision history
hm		27. apr. 2008	rev 1.0
	original version

*)
END_FUNCTION

(* POU JD2000, ST *)
FUNCTION JD2000 : REAL
VAR_INPUT
	DTI : DT;
END_VAR
VAR
END_VAR


(*
version 1.0	15. jul. 2008
programmer 	hugo
tested by	oscat

JULIAN calculates the astronomic julian date.

*)
JD2000 := DWORD_TO_REAL(DT_TO_DWORD(DTI) - 946728000) / 86400.0;



(* revision histroy
hm	15. jul. 2008	rev 1.0
	original release


*)	
END_FUNCTION

(* POU K_TO_C, ST *)
FUNCTION K_TO_C : REAL
VAR_INPUT
	Kelvin : REAL;
END_VAR
VAR
END_VAR

(*
version 1.0	4 dec 2006
programmer 	hugo
tested by		tobias

this function converts kelvin to celsius
*)
K_to_C := Kelvin + 273.15;
END_FUNCTION

(* POU KMH_TO_MS, ST *)
FUNCTION KMH_TO_MS : REAL
VAR_INPUT
	kmh : REAL;
END_VAR
VAR
END_VAR

(*
version 1.1	6 jan 2007
programmer 	hugo
tested by		tobias

this function converts velocities from Kilometers / hour to Meters / Second

*)
KMH_TO_MS := kmh * 0.2777777777777;

(* revision history
hm	4. feb 2007		rev 1.0
	original version

hm	6. jan 2008		rev 1.1
	improved performance

*)
END_FUNCTION

(* POU LANGEVIN, ST *)
FUNCTION LANGEVIN : REAL
VAR_INPUT
	X : REAL;
END_VAR
VAR
END_VAR

(*
version 1.1	11 mar 2008
programmer 	hugo
tested by		tobias

this function calculates the langevin function

*)
IF X = 0 THEN
	LANGEVIN := 0;
ELSE
	LANGEVIN := COTH(X) - 1/X;
END_IF;

(* revision history
hm	10.12.2007	rev 1.0
	original version

hm	11. mar 2008	rev 1.1
	changed formula to avoid problems when x = 0
*)
END_FUNCTION

(* POU LEAP_DAY, ST *)
FUNCTION LEAP_DAY : BOOL
VAR_INPUT
	IDATE : DATE;
END_VAR
VAR
END_VAR

(*
version 1.1	7. oct. 2008
programmer 	hugo
tested by	oscat


leap_day is true if the tested day is a leap day (29. of february).  
  
*)
LEAP_DAY := (MONTH_OF_DATE(idate) = 2) AND (DAY_OF_MONTH(idate) = 29);



(* change history

hm 	15. jun. 2008	rev 1.0
	original version

hm	7. oct. 2008	rev 1.1
	changed function month to month_of_date
*)
END_FUNCTION

(* POU LEGIONELLA, ST *)
FUNCTION_BLOCK LEGIONELLA
VAR_INPUT
	manual : BOOL;
	temp_boiler : REAL;
	temp_return : REAL := 100;
	DT_in: DT;
	rst : BOOL;
END_VAR
VAR_INPUT CONSTANT
	T_start: TOD := tod#03:00:00;
	day : INT := 7;
	temp_set : REAL := 70;
	temp_offset : REAL := 10;
	temp_hys : REAL := 5;
	t_max_heat: TIME := t#10m;
	t_max_ret : TIME := t#10m;
	tp_0: TIME := t#5m;
	tp_1: TIME := t#5m;
	tp_2: TIME := t#5m;
	tp_3: TIME := t#5m;
	tp_4: TIME := t#5m;
	tp_5: TIME := t#5m;
	tp_6: TIME := t#5m;
	tp_7: TIME := t#5m;
END_VAR
VAR_OUTPUT
	Heat : BOOL;
	pump : BOOL;
	valve0 : BOOL;
	valve1 : BOOL;
	valve2 : BOOL;
	valve3 : BOOL;
	valve4 : BOOL;
	valve5 : BOOL;
	valve6 : BOOL;
	valve7 : BOOL;
	run: BOOL;
	Status : BYTE;
END_VAR
VAR
	X1: timer_1;
	x2: sequence_8;
	x3: hyst_1;
	init: BOOL;
END_VAR

(*
version 1.2	23. oct 2008
programmer 	oscat
tested by	oscat

Legionella is a complete sequencer for up to 8 hot water lines that need to be sterilzed periodically.
legionella needs a DT input with the appropriate time, usually gererated by the rtc of the system. for system independence this time is connected externally.
T_start is the time when sterilazation should be started and day is the day_of_week when it should be performed (1=Monday and 7=sunday).
so sterilazation is autioimatically performed once a week at a specified time.
temp_set and temp_hys and temp_offset specify the boiler temperatur nedded for sterilization. as a defaut Temp_set is set to 70 deg C and Temp_hys is set to 5 deg C and temp_offset is 10 deg C.
a temp boiler input reads the boiler temperature of the hot water tank.
after a start pulse is gererated by the weekly timer or a manual test input the sequence is started:
1. the boiler is heated to temp_set + temp_offset + temp_hys = 85 deg C unless chaged at setup.
	the heat output is turned on and tells the heater to turn heating on. if the temp is not reached for a time of t_max_heat (10 min) the error output is set and the sequence is stopped.
2. after the specified temperature is reached, the output valve0 and pump is turned on and starts sterilization of line0 until temp_return has reached temp_set and continues to sterilize for a time of tp_0 (5 min default).
	if tmep_set is not reached at the temp_return_input then the error output is set and the sequence will be stopped.
	if there is no temp sensor for temp_return (the temperature at the return point for the circulation pump pls set this imput to a value greater then temp_set (by default use 100 deg C).
	in this case sterilization is performed for the default times without monitoring the return temp.
3. this sequence is repeated for up to valves.

connection scheme:

temp_boiler:	input oif the boiler temperature sensor.
temp_hys:		config value for the heater hysteresis, preset to 5 deg C.
temp_offset:	config value for the heater temp_offset against temp_set, preset to 10 deg C.
temp_set:		config value for the specified sterilization temperature, preset to 70 deg C.
temp_return:	input of the circulation return line temperature sensor, if not availabe set this value to 100 deg C.
manual:		manual input to start the sterilization by hand for diagnostic purposes, rising edge active, leave low for automatic operation.
DT_in:			date,time input supplied by a external real time clock.
T_start:		time of day when the sterilization should be started.
day:			config value for day of week when the process should be started, preset to sunday.
t_max_hest:	tmax time to be needed for the heater to heat the hot water tank to the specified value, preset to 10 min.

*)
(* startup initialization *)
IF NOT init THEN
	init := TRUE;
	X1.day := SHR(BYTE#128,day);
	X1.start := T_start;
	X3.low := Temp_offset + temp_set;
	X3.high := Temp_hys + X3.low;
	X2.wait0 := T_max_heat;
	X2.delay0 := TP_0;
	X2.delay1 := TP_1;
	X2.delay2 := TP_2;
	X2.delay3 := TP_3;
	X2.delay4 := TP_4;
	X2.delay5 := TP_5;
	X2.delay6 := TP_6;
	X2.delay7 := TP_7;
	X2.wait1 := T_max_ret;
	X2.wait2 := T_max_ret;
	X2.wait3 := T_max_ret;
	X2.wait4 := T_max_ret;
	X2.wait5 := T_max_ret;
	X2.wait6 := T_max_ret;
	X2.wait7 := T_max_ret;
	X2();
END_IF;

(* oerational code *)
X1(DTi := DT_in);
IF X1.Q OR manual OR x2.run THEN
	X3(in := temp_boiler);
	X2.in0 := X3.Q OR x3.win;
	X2.in1 := temp_return >= temp_set;
	X2.in2 := x2.in1;
	X2.in3 := x2.in1;
	X2.in4 := x2.in1;
	X2.in5 := x2.in1;
	X2.in6 := x2.in1;
	X2.in7 := x2.in1;
	X2.rst := rst;
	X2(start := X1.Q OR manual);
	run := x2.run;
	pump := x2.any;
	Heat := NOT X3.Q AND x2.run;
	valve0 := X2.Q0;
	valve1 := X2.Q1;
	valve2 := X2.Q2;
	valve3 := X2.Q3;
	valve4 := X2.Q4;
	valve5 := X2.Q5;
	valve6 := X2.Q6;
	valve7 := X2.Q7;
	pump := X2.any;
	status := X2.status;
ELSE;
	X2(start :=0);
	status := x2.status;
END_IF;

(* revision history

hm 17.jan 2007	rev 1.1
	rewritten to st for higher performance
	changes eeror output to esr compatible status output

hm	23. 10.2008	rev 1.2
	update code to use new version of timer_1
*)
END_FUNCTION_BLOCK

(* POU TIMER_1, ST *)
FUNCTION_BLOCK TIMER_1
VAR_INPUT
	E : BOOL := TRUE;
	DTI : DT;
	START : TOD;
	DURATION : TIME;
	DAY : BYTE := 2#0111_1111;
END_VAR
VAR_OUTPUT
	Q : BOOL;
END_VAR
VAR
	td : DATE;
	tdt : DT;
END_VAR

(*
version 2.1	6. nov. 2008
programmer 	oscat
tested by	oscat

this is a simple timer that generates an output pulse on selected days.
the output pulse width can be programmed with duration, if set to 0 no pulse is generated.
day specifies the specific days for the event to occur, bit 0 = sunday, bit 1 = saturday, bit 2 = friday ....
for all days to be active 127 has to be specified for DAY.

*)
td := DT_TO_DATE(DTI);
tdt := DATE_TO_DT(td) + TOD_TO_TIME(start);

Q := DTI >= tdt AND dti < tdt + duration AND E AND (SHR(BYTE#128, DAY_OF_WEEK(td)) AND day) > 0;



(*
1.12.2006 hm		rev 1.1
	corrected an error with pulse width = 0.

25.12.2006 hm		rev 1.2
	corrected an error when timer overflows.

14.apr 2007 hm		rev 1.3
	corrected an error while while output would not go active when start year would be 1970.
	increase accuracy by checking every 100ms
	added init section to compensate for timer overflow

15.9.2007 hm		rev 1.4
	replaced Time() with T_PLC_MS for compatibility and performance reasons

hm	1. okt 2007		rev 1.5
	corrected an error while output would not stay active over midnight.

hm	17. jan 2008	rev 1.6
	New code with better performance  
	Output is now only active during the time of day it is supposed to 
	no pulse is generated at power up

hm	7. oct. 2008	rev 1.7
	changed function weekday to day_of_week

hm	23. oct. 2008	rev 2.0
	new code, added input E, now days can be selected by bits in byte day

hm	6. nov. 2008	rev 2.1
	added default for input EN and input DAY
*)
END_FUNCTION_BLOCK

(* POU SEQUENCE_8, ST *)
FUNCTION_BLOCK SEQUENCE_8
VAR_INPUT
	in0 : BOOL := TRUE;
	in1 : BOOL := TRUE;
	in2 : BOOL := TRUE;
	in3 : BOOL := TRUE;
	in4 : BOOL := TRUE;
	in5 : BOOL := TRUE;
	in6 : BOOL := TRUE;
	in7 : BOOL := TRUE;
	start : BOOL;
	rst : BOOL;
	wait0 : TIME;
	delay0 : TIME;
	wait1 : TIME;
	delay1 : TIME;
	wait2 : TIME;
	delay2 : TIME;
	wait3 : TIME;
	delay3 : TIME;
	wait4 : TIME;
	delay4 : TIME;
	wait5 : TIME;
	delay5 : TIME;
	wait6 : TIME;
	delay6 : TIME;
	wait7 : TIME;
	delay7 : TIME;
END_VAR
VAR_INPUT CONSTANT
	stop_on_error : BOOL;
END_VAR
VAR_OUTPUT
	Q0 : BOOL;
	Q1 : BOOL;
	Q2 : BOOL;
	Q3 : BOOL;
	Q4 : BOOL;
	Q5 : BOOL;
	Q6 : BOOL;
	Q7 : BOOL;
	any : BOOL;
	run: BOOL;
	step : INT := -1;
	status : BYTE;
END_VAR
VAR
	last : TIME;
	edge : BOOL;
	tx: TIME;
	init: BOOL;
END_VAR

(*
version 1.4	17 sep 2007
programmer 	oscat
tested by		hans

sequence_8 enables run when a low to high transition is present on start.
a low to high transition on start will restart the sequencer at any time while a rst will hold the sequencer in reset while true.
after run is enabled with a rising edge on start the sequencer waits for wait0 on in0 to enable q0 which stays on for delay0.
the next cycle starts with wait1, continues with delay 1 and so on...
if an edge is not detected during the wait period, the sequencer will then display the error number on the status output.
The status numbers are 1 .. 8 for erros in step 0..7.
after the last step that sets q7, the sequencer leaves q7 on for delay7 and then resets to the initial state.
a step output will indicate the current step of the sequencer and will also be present with a fault condition.
after the first output is turened on the sequencer switches from q0 to q1 and so on, at any time there is only one output enabled.
if an input signal is not detected during a wait period, the sequencer will display the error number ( 1 for in0, 2 for in1 .... ).
when an error is present and the config variable stop_on_error is set then the sequencer will stop. otherwise it will continue.
The status output will also display 110 for waiting and 111 sequece running.

*)
(* read sps timer *)
tx := DWORD_TO_TIME(T_PLC_MS());

(* initialize on startup *)
IF NOT init THEN
	last := tx;
	init := TRUE;
	status := 110;
END_IF;

(* asynchronous reset *)
IF rst THEN
	step := -1;
	Q0 := 0;
	Q1 := 0;
	Q2 := 0;
	Q3 := 0;
	Q4 := 0;
	Q5 := 0;
	Q6 := 0;
	Q7 := 0;
	status := 110;
	run := 0;

(* edge on start input restarts the sequencer *)
ELSIF start AND NOT edge THEN
	step := 0;
	last := tx;
	status := 111;
	Q0 := 0;
	Q1 := 0;
	Q2 := 0;
	Q3 := 0;
	Q4 := 0;
	Q5 := 0;
	Q6 := 0;
	Q7 := 0;
	run := 1;
END_IF;
edge := start;

(* check if stop on error is necessary *)
IF status > 0 AND status < 100 AND stop_on_error THEN RETURN; END_IF;

(* sequence is running *)
IF run AND step = 0 THEN
	IF NOT q0 AND in0 AND tx - last <= wait0 THEN
		Q0 := TRUE;
		last := tx;
	ELSIF NOT q0 AND tx - last > wait0 THEN
		status := 1;
		run := FALSE;
	ELSIF q0 AND tx - last >= delay0 THEN
		step := 1;
		last := tx;
	END_IF;
END_IF;
IF run AND step = 1 THEN
	IF NOT q1 AND in1 AND tx - last <= wait1 THEN
		Q0 := FALSE;
		Q1 := TRUE;
		last := tx;
	ELSIF NOT q1 AND Tx - last > wait1 THEN
		status := 2;
		q0 := FALSE;
		run := FALSE;
	ELSIF q1 AND tx - last >= delay1 THEN
		step := 2;
		last := tx;
	END_IF;
END_IF;
IF run AND step = 2 THEN
	IF NOT q2 AND in2 AND tx - last <= wait2 THEN
		Q1 := FALSE;
		Q2 := TRUE;
		last := tx;
	ELSIF NOT q2 AND Tx - last > wait2 THEN
		status := 3;
		q1 := FALSE;
		run := FALSE;
	ELSIF q2 AND tx - last >= delay2 THEN
		step := 3;
		last := tx;
	END_IF;
END_IF;
IF run AND step = 3 THEN
	IF NOT q3 AND in3 AND tx - last <= wait3 THEN
		Q2 := FALSE;
		Q3 := TRUE;
		last := tx;
	ELSIF NOT q3 AND Tx - last > wait3 THEN
		status := 4;
		q2 := FALSE;
		run := FALSE;
	ELSIF q3 AND tx - last >= delay3 THEN
		step := 4;
		last := tx;
	END_IF;
END_IF;
IF run AND step = 4 THEN
	IF NOT q4 AND in4 AND tx - last <= wait4 THEN
		Q3 := FALSE;
		Q4 := TRUE;
		last := tx;
	ELSIF NOT q4 AND Tx - last > wait4 THEN
		status := 5;
		q3 := FALSE;
		run := FALSE;
	ELSIF q4 AND tx - last >= delay4 THEN
		step := 5;
		last := tx;
	END_IF;
END_IF;
IF run AND step = 5 THEN
	IF NOT q5 AND in5 AND tx - last <= wait5 THEN
		Q4 := FALSE;
		Q5 := TRUE;
		last := tx;
	ELSIF NOT q5 AND Tx - last > wait5 THEN
		status := 6;
		q4 := FALSE;
		run := FALSE;
	ELSIF q5 AND tx - last >= delay5 THEN
		step := 6;
		last := tx;
	END_IF;
END_IF;
IF run AND step = 6 THEN
	IF NOT q6 AND in6 AND tx - last <= wait6 THEN
		Q5 := FALSE;
		Q6 := TRUE;
		last := tx;
	ELSIF NOT q6 AND Tx - last > wait6 THEN
		status := 7;
		q5 := FALSE;
		run := FALSE;
	ELSIF q6 AND tx - last >= delay6 THEN
		step := 7;
		last := tx;
	END_IF;
END_IF;
IF run AND step = 7 THEN
	IF NOT q7 AND in7 AND tx - last <= wait7 THEN
		Q6 := FALSE;
		Q7 := TRUE;
		last := tx;
	ELSIF NOT q7 AND Tx - last > wait7 THEN
		status := 8;
		q6 := FALSE;
		run := FALSE;
	ELSIF q7 AND tx - last >= delay7 THEN
		step := -1;
		Q7 := FALSE;
		Run := FALSE;
		status := 110;
	END_IF;
END_IF;
any := q0 OR q1 OR q2 OR q3 OR q4 OR q5 OR q6 OR q7;

(*
hm 1.10.06		rev 1.1
	corrected delay logic to be after event and not before
	added any output

hm 1.12.06		rev 1.2
	corrected failure in sequence logic.
	added init at startup to prevent from initial statuss after start.

hm 17.1.2007		rev 1.3
	changed output fault to status for better compatibility with other modules (ESR)
	added stop on error functionality and setup variable
	default for inputs in0..7 is true.
	renames variable state to step

hm	17.sep 2007		rev 1.4
	replaced time() with T_PLC_MS() for compatibility reasons

*)
END_FUNCTION_BLOCK

(* POU LIST_CLEAN, ST *)
FUNCTION LIST_CLEAN : BOOL
VAR_INPUT
	SEP : BYTE;
END_VAR
VAR_IN_OUT
	LIST : STRING(255);
END_VAR
VAR
	pt : POINTER TO ARRAY[1..255] OF BYTE;
	pos: INT;
	pw : INT;
	last: BYTE;
	c: BYTE;
END_VAR


(*
version 1.0	28. jun. 2008
programmer 	hugo
tested by	oscat

LIST_CLEAN bereinigt eine liste von leeren Elementen.
die liste liegt als string von elementen vor die mit den zeichen SEP separiert sind.

*)
pt := ADR(LIST);

last := sep;
REPEAT
   pos := pos + 1;
   c := pt^[pos];
   IF last <> sep OR c <> sep THEN
      pw := pw + 1;
      pt^[pw] := c;
   END_IF;
   last := c;
UNTIL pos > 254 OR c = 0
END_REPEAT;

IF pw > 1 THEN
  pw := pw - 1;
  IF pt^[pw] = sep THEN pt^[pw] := 0; END_IF;
END_IF;

(* retrun TRUE *)
LIST_CLEAN := TRUE;



(* revision histroy
hm	28. jun. 2008	rev 1.0
	original release


*)	
END_FUNCTION

(* POU LIST_GET, ST *)
FUNCTION LIST_GET : STRING(STRING_LENGTH)
VAR_INPUT
	SEP : BYTE;
	POS : INT;
END_VAR
VAR_IN_OUT
	LIST : STRING(255);
END_VAR
VAR
	i : INT := 1;
	o : INT := 1;
	pt : POINTER TO ARRAY[1..255] OF BYTE;
	po : POINTER TO ARRAY[1..STRING_LENGTH] OF BYTE;
	cnt: INT;
	c: BYTE;
END_VAR


(*
version 1.0	20. jun 2008
programmer 	hugo
tested by	oscat

LIST_GET liefert das element an der stelle pos einer liste.
die liste liegt als string von elementen vor die mit den zeichen SEP separiert sind.

*)
(* load pointers *)
pt := ADR(LIST);
po := ADR(LIST_GET);

(* search for the n-th occurence of a separation character and store position in i *)
WHILE (cnt < pos) AND (i < 255) AND (pt^[i] > 0) DO
	IF pt^[i] = sep THEN cnt := cnt + 1; END_IF;
	i := i + 1;
END_WHILE

(* copy the list element to output *)
IF i < 255 THEN c := pt^[i]; END_IF;
WHILE (c <> sep) AND (c > 0) AND (o < string_length) AND (i < 255) DO
	po^[o] :=pt^[i];
	o := o + 1;
	i := i + 1;
	c := pt^[i];
END_WHILE;

(* terminate the output string *)
po^[o] := 0;



(* revision histroy
hm	20. jun. 2008	rev 1.0
	original release


*)	
END_FUNCTION

(* POU LIST_INSERT, ST *)
FUNCTION LIST_INSERT : BOOL
VAR_INPUT
	SEP : BYTE;
	POS : INT;
	INS : STRING(STRING_LENGTH);
END_VAR
VAR_IN_OUT
	LIST : STRING(255);
END_VAR
VAR
	i : INT;
	pt : POINTER TO ARRAY[1..255] OF BYTE;
	cnt : INT;
	c : BYTE;
	tmp : STRING(STRING_LENGTH);
END_VAR


(*
version 1.1	17. dec. 2008
programmer 	hugo
tested by	oscat

LIST_INSERT setzt ein element an der stelle pos in eine liste ein.
die liste liegt als string von elementen vor die mit den zeichen SEP separiert sind.

*)
(* load pointers *)
pt := ADR(LIST);

(* search for the n-th occurence of a separation character and store position in i *)
c := pt^[1];
WHILE (cnt < pos) AND (i < 255) AND (c > 0) DO
	i := i + 1;
	c := pt^[i];
	IF c = sep THEN cnt := cnt + 1; END_IF;
END_WHILE;

(* copy the new element into the list *)
tmp := CHR_TO_STRING(SEP);
IF i = 0 THEN
	tmp := CONCAT(INS,tmp);
	LIST := INSERT(LIST, tmp, 0);
ELSE
	tmp := CONCAT(tmp, INS);
	LIST := INSERT(LIST, tmp, i - 1);
END_IF;


LIST_INSERT := TRUE;



(* revision histroy
hm	28. jun. 2008	rev 1.0
	original release

hm	17. dec. 2008	rev 1.1
	changes name of function chr to chr_to_string

*)	
END_FUNCTION

(* POU LIST_LEN, ST *)
FUNCTION LIST_LEN : INT
VAR_INPUT
	SEP : BYTE;
END_VAR
VAR_IN_OUT
	LIST : STRING(255);
END_VAR
VAR
	pt : POINTER TO ARRAY[1..255] OF BYTE;
	l: INT;
	pos: INT;
END_VAR


(*
version 1.1	16. oct. 2008
programmer 	hugo
tested by	oscat

LIST_LEN liefert die anzahl der elemente einer liste.
die liste liegt als string von elementen vor die mit den zeichen SEP separiert sind.

*)
PT := ADR(LIST);
LIST_LEN := 1;
l := LEN(list);
FOR pos := 1 TO l DO
	IF pt^[pos] = SEP THEN LIST_LEN := LIST_LEN + 1; END_IF;
END_FOR;



(* code before rev 1.1
LIST_LEN := COUNT_CHAR(LIST, SEP) + 1;
*)


(* revision histroy
hm	25. jun. 2008	rev 1.0
	original release

hm	16. oct. 2008	rev 1.1
	fixed a problem where list_len would only work up to STRING_LENGTH

*)	
END_FUNCTION

(* POU LIST_NEXT, ST *)
FUNCTION_BLOCK LIST_NEXT
VAR_INPUT
	SEP : BYTE;
	RST : BOOL;
END_VAR
VAR_IN_OUT
	LIST : STRING(255);
END_VAR
VAR_OUTPUT
	LEL : STRING(STRING_LENGTH);
	NUL : BOOL;
END_VAR
VAR
	pt : POINTER TO ARRAY[1..255] OF BYTE;
	stop: INT;
	start: INT;
	pos : INT := 1;
END_VAR


(*
version 1.0	25. jun. 2008
programmer 	hugo
tested by	oscat

LIST_NEXT retrieves the next element of a list, starting from element 0 after reset or first init.
when the end of the lisat is reached a '' empty string is returned and NUL is set to true.
die liste liegt als string von elementen vor die mit den zeichen SEP separiert sind.

*)
(* load pointers *)
pt := ADR(LIST);
stop := LEN(LIST);

IF rst THEN
	start := 0;
	pos := 1;
	NUL := FALSE;
END_IF;

(* search next occurence of separation character or end of list *)
WHILE pos <= stop DO
	IF pt^[pos] = SEP THEN EXIT; END_IF;
	pos := pos + 1;
END_WHILE;
IF start <= stop THEN
	LEL := MID(LIST, pos - start - 1, start + 1);
	start := pos;
	pos := pos + 1;
ELSE
	LEL := '';
	NUL := TRUE;
END_IF;



(* revision histroy
hm	25. jun. 2008	rev 1.0
	original release


*)	
END_FUNCTION_BLOCK

(* POU LIST_RETRIEVE, ST *)
FUNCTION LIST_RETRIEVE : STRING(STRING_LENGTH)
VAR_INPUT
	SEP : BYTE;
	POS : INT;
END_VAR
VAR_IN_OUT
	LIST : STRING(255);
END_VAR
VAR
	i,o : INT;
	pt : POINTER TO ARRAY[0..255] OF BYTE;
	po : POINTER TO ARRAY[0..STRING_LENGTH] OF BYTE;
	cnt: INT;
	c: BYTE;
	p : INT;
	l: INT;
END_VAR


(*
version 1.0	28. jun 2008
programmer 	hugo
tested by	oscat

LIST_RETRIEVE liefert das element an der stelle pos einer liste und löscht das element aus der liste.
die liste liegt als string von elementen vor die mit den zeichen SEP separiert sind.

*)
(* load pointers *)
pt := ADR(LIST);
po := ADR(LIST_RETRIEVE);
l := LEN(LIST);

(* search for the n-th occurence of a separation character and store position in i *)
WHILE (cnt < pos) AND (i < 255) AND (pt^[i] > 0) DO
	IF pt^[i] = sep THEN cnt := cnt + 1; END_IF;
	i := i + 1;
END_WHILE

p := i;	(* store position for deletion in list *)

(* copy the list element to output *)
IF i < 255 THEN c := pt^[i]; END_IF;
WHILE (c <> sep) AND (c > 0) AND (o < string_length) AND (i < 255) DO
	po^[o] :=pt^[i];
	o := o + 1;
	i := i + 1;
	c := pt^[i];
END_WHILE;

IF cnt = pos THEN
	IF i = L THEN
		LIST := LEFT(LIST, p - 1);
	ELSE
		LIST := DELETE(LIST, i - p + 1, p + 1);
	END_IF;
END_IF;


(* terminate the output string *)
po^[o] := 0;



(* revision histroy
hm	28. jun. 2008	rev 1.0
	original release


*)	
END_FUNCTION

(* POU LIST_RETRIEVE_MAX, ST *)
FUNCTION LIST_RETRIEVE_MAX : STRING(STRING_LENGTH)
VAR_INPUT
	SEP : BYTE;
END_VAR
VAR_IN_OUT
	LIST : STRING(255);
END_VAR
VAR
	pt : POINTER TO ARRAY[1..255] OF BYTE;
	l: INT;
	pos: INT;
	last: INT;
	lx: INT;
	mpos: INT := 1;
END_VAR


(*
version 1.0	22. oct. 2008
programmer 	hugo
tested by	oscat

LIST_MAX liefert das längste elemente einer liste.
die liste liegt als string von elementen vor die mit den zeichen SEP separiert sind.

*)
PT := ADR(LIST);
l := LEN(list);
FOR pos := 1 TO l DO
	IF pt^[pos] = sep THEN
		IF pos - last - 1 > lx THEN
			mpos := last + 1;
			lx := pos - last - 1;
		END_IF;
		last := pos;
	END_IF;
END_FOR;

(* check length of last element *)
IF l - last > lx THEN
	mpos := last + 1;
	lx := l - last;
	LIST_RETRIEVE_MAX := RIGHT(list, lx);
	list := LEFT(list, last - 1);
ELSE
	LIST_RETRIEVE_MAX := MID(LIST, lx, mpos);
	LIST := DELETE(LIST, lx + 1, mpos);
END_IF;



(* revision histroy
hm	22. oct. 2008	rev 1.0
	original release


*)	
END_FUNCTION

(* POU LIST_RETRIEVE_MIN, ST *)
FUNCTION LIST_RETRIEVE_MIN : STRING(STRING_LENGTH)
VAR_INPUT
	SEP : BYTE;
END_VAR
VAR_IN_OUT
	LIST : STRING(255);
END_VAR
VAR
	pt : POINTER TO ARRAY[1..255] OF BYTE;
	l: INT;
	pos: INT;
	last: INT;
	lx: INT;
	mpos: INT := 1;
END_VAR


(*
version 1.0	23. oct. 2008
programmer 	hugo
tested by	oscat

LIST_MAX liefert das längste elemente einer liste.
die liste liegt als string von elementen vor die mit den zeichen SEP separiert sind.

*)
PT := ADR(LIST);
l := LEN(list);
lx := 255;
FOR pos := 1 TO l DO
	IF pt^[pos] = sep THEN
		IF pos - last - 1 < lx THEN
			mpos := last + 1;
			lx := pos - last - 1;
			(* if we found an element with length 0 then we can stop *)
		END_IF;
		last := pos;
		IF lx = 0 THEN EXIT; END_IF;
	END_IF;
END_FOR;

(* check length of last element *)
IF l - last < lx THEN
	mpos := last + 1;
	lx := l - last;
	LIST_RETRIEVE_MIN := RIGHT(list, lx);
	list := LEFT(list, last - 1);
ELSE
	LIST_RETRIEVE_MIN := MID(LIST, lx, mpos);
	LIST := DELETE(LIST, lx + 1, mpos);
END_IF;



(* revision histroy
hm	23. oct. 2008	rev 1.0
	original release


*)	
END_FUNCTION

(* POU LIST_SORT_L, ST *)
FUNCTION LIST_SORT_L : STRING(255)
VAR_INPUT
	SEP : BYTE;
END_VAR
VAR_IN_OUT
	LIST : STRING(255);
END_VAR
VAR
	element: STRING(STRING_LENGTH);
	sepx: STRING(1);
END_VAR


(*
version 1.1	17. dec. 2008
programmer 	hugo
tested by	oscat

LIST_SORT_L liefert eine Liste die nach Länge der elemente sortiert ist.
die liste liegt als string von elementen vor die mit den zeichen SEP separiert sind.

*)
sepx := CHR_TO_STRING(sep);
WHILE list <> '' DO
	IF list = sepx THEN
		LIST_SORT_L := CONCAT(sepx, LIST_SORT_L);
		list := '';
		RETURN;
	ELSE
		element := LIST_RETRIEVE_MIN(SEP,LIST);
		LIST_SORT_L := CONCAT(LIST_SORT_L, element);
		LIST_SORT_L := CONCAT(LIST_SORT_L, sepx);
	END_IF;
END_WHILE;
(* delete the last separation character *)
LIST_SORT_L := LEFT(LIST_SORT_L, LEN(LIST_SORT_L) - 1);


(* revision histroy
hm	23. oct. 2008	rev 1.0
	original release

hm	17. dec. 2008	rev 1.1
	changes name of function chr to chr_to_string

*)	
END_FUNCTION

(* POU LTCH, ST *)
FUNCTION_BLOCK LTCH
VAR_INPUT
	D : BOOL;
	L : BOOL;
	RST : BOOL;
END_VAR
VAR_OUTPUT
	Q : BOOL;
END_VAR
VAR
END_VAR

(*
version 1.2	30. oct. 2008
programmer 	hugo
tested by	oscat

Transparent Latch with asynchronous reset


*)
(* as long as L is true, the latch is transparent and and change of D is transferred to Q *)
(* of course only when there is no asynchronous reset *)
IF rst THEN				(* if asynchronous reset then Q=0 *)
	Q := FALSE;
ELSIF L THEN			(* latch is transparent *)
	Q := D;
END_IF;


(* revision history
hm	4. aug 2006		rev 1.0
	original version

hm	27. dec 2007	rev 1.1
	changed code for better performance

hm	30. oct. 2008	rev 1.2
	deleted unnecessary init with 0

*)
END_FUNCTION_BLOCK

(* POU LTCH_4, ST *)
FUNCTION_BLOCK LTCH_4
VAR_INPUT
	D0 : BOOL;
	D1 : BOOL;
	D2 : BOOL;
	D3 : BOOL;
	L : BOOL;
	RST : BOOL;
END_VAR
VAR_OUTPUT
	Q0 : BOOL;
	Q1 : BOOL;
	Q2 : BOOL;
	Q3 : BOOL;
END_VAR
VAR
END_VAR

(*
version 1.2	30. oct. 2008
programmer 	hugo
tested by	oscat

Quad Transparent Latch with asynchronous reset


*)
(* as long as L is true, the latch is transparent and and change of D is transferred to Q *)
(* of course only when there is no asynchronous reset *)
IF rst THEN				(* if asynchronous reset then Q=0 *)
	Q0 := Q1 := Q2 := Q3 := FALSE;
ELSIF L THEN			(* latch is transparent *)
	Q0 := D0;
	Q1 := D1;
	Q2 := D2;
	Q3 := D3;
END_IF;

(* revision history
hm	4. aug 2006		rev 1.0
	original version

hm	27. dec 2007	rev 1.1
	changed code for better performance

hm	30. oct. 2008	rev 1.2
	deleted unnecessary init with 0
*)
END_FUNCTION_BLOCK

(* POU LTIME_TO_UTC, ST *)
FUNCTION LTIME_TO_UTC : DT
VAR_INPUT
	LTIME : DT;
	DST : BOOL;
	TIME_ZONE_OFFSET : INT;
END_VAR
VAR
END_VAR

(*
version 1.5	20. oct. 2008
programmer 	hugo
tested by	oscat

LTIME_TO_UTC calculates UTC (World Time) from a local time LTIME. utc is calculated 
by subtracting Time_Zone_Offset from ltime and if dst it true subtracting an additional hour from ltime.

*)
LTIME_TO_UTC := DWORD_TO_DT(DT_TO_DWORD(Ltime) - time_zone_offset * 60 - BOOL_TO_INT(DST)*3600);


(* revision history
hm 5.7.2007		rev 1.0		
	original version

hm 5.11.2007		rev 1.1
	replaced literal constant with variable because of error in möller ecp4 compiler

hm	12.nov 2007	rev 1.2
	changed Type of time_zone_offset from time to int to allow for time zones with negative offset

hm	8. dec 2007	rev 1.3
	corrected a problem with time_zone_offset

hm	14. oct. 2008	rev 1.4
	changed time_zone_offset from int to real to allow for half hour offset

hm	20. oct. 2006	rev 1.5
	changed time_zone_offset from Real to INT, now in Minutes

*)
END_FUNCTION

(* POU M_D, ST *)
FUNCTION_BLOCK M_D
VAR_INPUT
	start : BOOL;
	stop : BOOL;
	tmax : TIME := t#10d;
	rst: BOOL;
END_VAR
VAR_OUTPUT
	PT : TIME;
	ET : TIME;
	run : BOOL;
END_VAR
VAR
	edge : BOOL := 0;
	T0 : TIME;
	tx: TIME;
	startup: BOOL;
END_VAR

(*
	version 1.1	16 sep 2007
	programmer 	hugo
	tested BY		tobias

m_d measures the time between a rising edge on start to a rising edge on stop and returs the last measured value on the output PT.
a second output ET is starting from 0 at the rising edge of start and is counting up until the rising edge of stop occurs.
the asynchronous input rst can reset the outputs at any time.
tmax defines a timeout wich is the maximum measurable time between start and stop, if this time is exceeded the outputs will stay at 0.
*)
(* check for rst input *)
IF rst OR et >= tmax THEN
	pt := t#0ms;
	et := t#0ms;
	startup := FALSE;
	run := FALSE;
END_IF;

(* avoid timers to start when input is true at startup *)
IF NOT startup THEN
	edge := start;
	startup := TRUE;
END_IF;

(* read system timer *)
tx := DWORD_TO_TIME(T_PLC_MS());

(* detect rising edge on start *)
IF start AND NOT edge AND NOT stop THEN
	t0 := tx;
	run := TRUE;
	pt := t#0s;
ELSIF stop AND run THEN
	pt := et;
	run := FALSE;
END_IF;
edge := start;
IF run THEN et := tx - t0; END_IF;

(* revision history
hm		2.5.2007	rev 1.0
	original version

hm		16.9.2007	rev 1.1
	changes time() to T_plc_ms() for compatibility reasons

*)
END_FUNCTION_BLOCK

(* POU M_T, ST *)
FUNCTION_BLOCK M_T
VAR_INPUT
	IN : BOOL;
	TMAX : TIME := t#10d;
	RST : BOOL;
END_VAR
VAR_OUTPUT
	PT : TIME;
	ET: TIME;
END_VAR
VAR
	edge : BOOL;
	start : TIME;
	tx: TIME;
END_VAR

(*
	version 1.3	17. dec. 2008
	programmer 	hugo
	tested BY	oscat

m_t measures the with of a high pulse and returs the last measured pulse width on output PT.
a second output ET is starting from 0 at the rising edge and counting up until the falling edge occurs and resetts et to 0.
the asynchrtonous input rst can reset the outputs at any time.
tmax defines a maximum measurable time, if this value is exceeded the outputs will be reset to 0.
*)
(* read system time *)
tx := DWORD_TO_TIME(T_PLC_MS());

IF RST OR ET >= TMAX THEN
	PT := ET := t#0s;
ELSIF IN THEN
	IF NOT edge THEN start := tx; END_IF;
	ET := tx - start;
ELSE
	PT := ET;
END_IF;
edge := IN;


(* code for rev 1.2

(* check for rst input *)
IF rst OR et >= tmax THEN
	init := FALSE;
	startup := FALSE;
	pt := t#0ms;
	et := t#0ms;
END_IF;

(* avoid timers to start when input is true at startup *)
IF NOT startup THEN
	edge := in;
	startup := TRUE;
END_IF;

(* read system timer *)
tx := DWORD_TO_TIME(T_PLC_MS());

(* edge trigger rising and falling edge *)
IF in XOR edge THEN
	edge := in;
	(* rising edge starts measurement *)
	IF in THEN
		init := TRUE;
		start := Tx;
	(* falling edge stops measurement *)
	ELSIF init THEN
		stop := Tx;
		pt := stop - start;
	END_IF;
END_IF;

IF init AND in THEN
	et := Tx - start; ELSE et := t#0ms;
END_IF;
*)




(* revision history
hm	4. aug. 2006	rev 1.0
	original version

hm	2. may. 2007	rev 1.1
	added init variable to avoid unreasonable measurement if falling edge occurs first.
	added et (elapsed time) output to count from 0 at rising edge until a falling edge resets et to 0.
	added reset input.

hm	16. sep. 2007	rev 1.2
	changes time() to T_plc_ms() for compatibility reasons

hm	17. dec. 2008	rev 1.3
	code optimized

*)
END_FUNCTION_BLOCK

(* POU M_TX, ST *)
FUNCTION_BLOCK M_TX
VAR_INPUT
	in: BOOL;
	tmax : TIME := t#10d;
	rst : BOOL;
END_VAR
VAR_OUTPUT
	TH : TIME;
	TL : TIME;
	DC : REAL;
	F: REAL;
	ET : TIME;
END_VAR
VAR
	edge : BOOL := 0;
	start: TIME;
	stop:TIME;
	tx: TIME;
	rise : BOOL;
	fall : BOOL;
	startup: BOOL;
END_VAR

(*
	version 1.2	16 sep 2007
	programmer 	oscat
	tested BY		oscat

this measures the timing of a signal
TH is the high pulse width
TL is the low pulse width
DC is the duty cycle
F is the frequency
ET will start at 0 with a rising edge and count up till the next rising edge starts from 0 again. 
the acuracy depends on the cycle time of the sps and is limited to 1ms resolution.
an asynchronous reset can reset all outputs to 0 at any time.
the input tmax can configure a timeout for ET where the function block will outomatically reset itself.
tmx is predefined to 10 days.
*)
(* check FOR rst input *)
IF rst OR (et >= tmax) THEN
	rise := FALSE;
	fall := FALSE;
	startup := FALSE;
	th := t#0ms;
	tl := t#0ms;
	DC := 0;
	F := 0;
	ET := t#0s;
END_IF;

(* avoid timers to start when input is true at startup *)
IF NOT startup THEN
	edge := in;
	startup := TRUE;
END_IF;

(* read system timer *)
tx := DWORD_TO_TIME(T_PLC_MS());

(* edge trigger rising and falling edge *)
IF in XOR edge THEN
	edge := in;
	(* rising edge starts measurement *)
	IF in THEN
		start := Tx;
		rise := TRUE;
		IF fall THEN tl := start - stop; END_IF;
		IF th > t#0ms AND tl > t#0ms THEN
			dc := TIME_TO_REAL(th) / TIME_TO_REAL(th+tl);
			f := 1000 / TIME_TO_REAL(th + tl);
		END_IF;
	(* falling edge starts second cycle measurement *)
	ELSE
		stop := Tx;
		fall := TRUE;
		IF rise THEN th := stop - start; END_IF;
		IF th > t#0ms AND tl > t#0ms THEN
			dc := TIME_TO_REAL(th) /  TIME_TO_REAL(th+tl);
			f := 1000 / TIME_TO_REAL(th + tl);
		END_IF;
	END_IF;
END_IF;
IF rise THEN et := tx - start; END_IF;

(* revision history
hm		4. aug 2006	rev 1.0
	original version

hm		2. mai 2007	rev 1.1
	made sure that no undefined values would be measured at startup conditions
	added output et
	added rst input
	added tmax input

hm		16.9.2007	rev 1.2
	changes time() to T_plc_ms() for compatibility reasons

*)
END_FUNCTION_BLOCK

(* POU MANUAL_1, ST *)
FUNCTION_BLOCK MANUAL_1
VAR_INPUT
	IN : BOOL;
	MAN : BOOL;
	M_I : BOOL;
	SET : BOOL;
	RST : BOOL;
END_VAR
VAR_OUTPUT
	Q : BOOL;
	STATUS : BYTE;
END_VAR
VAR
	S_edge : BOOL;
	r_edge : BOOL;
	edge: BOOL;
END_VAR

(*
version 1.1	17. oct. 2008
programmer 	hugo
tested by	oscat

MANUAL_1 is a manual override for digital signals.
When MAN = FALSE, the output follows IN and when MAN = TRUE the Output follows M_I.


*)
IF NOT man THEN
	Q := IN;
	STATUS := 100;
	edge := FALSE;
ELSIF NOT s_edge AND set THEN
	Q := edge := TRUE;
	status := 101;
ELSIF NOT r_edge AND rst THEN
	Q := FALSE;
	edge := TRUE;
	status := 102;
ELSIF NOT edge THEN
	Q := M_I;
	status := 103;
END_IF;

(* remember levels of manual signals *)
s_edge := SET;
r_edge := RST;



(* revision history
hm	17. jun 2008	rev 1.0
	original version

hm	17. oct 2008	rev 1.1
	deleted unnecessary variable m_edge
*)
END_FUNCTION_BLOCK

(* POU MANUAL_2, ST *)
FUNCTION_BLOCK MANUAL_2
VAR_INPUT
	IN : BOOL;
	ENA : BOOL;
	ON : BOOL;
	OFF : BOOL;
	MAN : BOOL;
END_VAR
VAR_OUTPUT
	Q : BOOL;
	STATUS : BYTE;
END_VAR
VAR
END_VAR

(*
version 1.0	22. sep. 2008
programmer 	hugo
tested by	oscat

MANUAL_2 is a manual override for boolean signals.
it has static force high and low as well as a manual input.

*)
IF ena THEN
	IF NOT ON AND NOT OFF THEN
		Q := IN;
		STATUS := 100;
	ELSIF on AND NOT off THEN
		Q := TRUE;
		STATUS := 101;
	ELSIF NOT on AND off THEN
		q := FALSE;
		STATUS := 102;
	ELSE
		Q := MAN;
		STATUS := 103;
	END_IF;
ELSE
	Q := FALSE;
	STATUS := 104;
END_IF;



(* revision history
hm	22. sep. 2008		rev 1.0
	original version

*)
END_FUNCTION_BLOCK

(* POU MANUAL_4, ST *)
FUNCTION_BLOCK MANUAL_4
VAR_INPUT
	I0, I1, I2, I3 : BOOL;
	MAN : BOOL;
	STP : BOOL;
	M0, M1, M2, M3 : BOOL;
END_VAR
VAR_OUTPUT
	Q0, Q1, Q2, Q3 : BOOL;
	STATUS : BYTE;
END_VAR
VAR
	edge: BOOL;
	pos : INT;
	tog: BOOL;
END_VAR


(*
version 1.0	17. jun 2008
programmer 	hugo
tested by	oscat

MANUAL_4 is a manual override for digital signals.
When MAN = FALSE, the output follows IN and when MAN = TRUE the Output follows M_I.


*)
IF man THEN
	IF NOT TOG THEN
		Q0 := M0;
		Q1 := M1;
		Q2 := M2;
		Q3 := M3;
		STATUS := 101;
	END_IF;
	IF STP AND NOT edge THEN
		tog := TRUE;
		CASE pos OF
			0:	Q0 := TRUE;
				Q1 := FALSE;
				Q2 := FALSE;
				Q3 := FALSE;
				STATUS := 110;
			1:	Q0 := FALSE;
				Q1 := TRUE;
				Q2 := FALSE;
				Q3 := FALSE;
				STATUS := 111;
			2:	Q0 := FALSE;
				Q1 := FALSE;
				Q2 := TRUE;
				Q3 := FALSE;
				STATUS := 112;
			3:	Q0 := FALSE;
				Q1 := FALSE;
				Q2 := FALSE;
				Q3 := TRUE;
				STATUS := 113;
		END_CASE;
		pos := INC(pos,1,3);
	END_IF;
ELSE
	Q0 := I0;
	Q1 := I1;
	Q2 := I2;
	Q3 := I3;
	STATUS := 100;
	tog := FALSE;
	pos := 0;
END_IF;

(* remember status of stp *)
edge := STP;



(* revision history
hm	17. jun 2008		rev 1.0
	original version

*)
END_FUNCTION_BLOCK

(* POU MATRIX, ST *)
FUNCTION_BLOCK MATRIX
VAR_INPUT
	x1, x2, x3, x4, X5 : BOOL;
END_VAR
VAR_INPUT CONSTANT
	Release : BOOL;
END_VAR
VAR_OUTPUT
	code : BYTE;
	TP : BOOL;
	y1: BOOL := TRUE;
	y2, y3, y4 : BOOL;
END_VAR
VAR
	line : BYTE;
	X : ARRAY[0..3] OF BYTE; (* scan line inputs *)
	L : ARRAY[0..3] OF BYTE; (* scan line status *)
	i: INT;
	temp: BYTE;
END_VAR

(*
version 1.3	26 oct. 2008
programmer 	hugo
tested by	oscat

MATRIX is a matrix keyboard encoder for 4 rows and up to 5 columns.
matrix can send a code while a key is pressed and it sends another code while a key is released when the setup variable 'release' is set to true.
the setup variable release is false the code is only sent when the key is pressed.
the output byte holds the 5 columns in the lowest bits 0..2  and the row number in bits 4..6, while bit 7 is true for a key pressed and false for a key released.

*)
TP := FALSE;
CODE := 0;
(* read scan lines *)
X[line].0 := X1;
X[line].1 := X2;
X[line].2 := X3;
X[line].3 := X4;
X[line].4 := X5;

(* compare for change *)
FOR i := 0 TO 3 DO
	IF X[i] <> L[i] THEN
		(* scan line information has changed code need to be found and generated *)
		temp := x[i] XOR L[i];
		IF temp.0 THEN
			CODE := 1;
			code.7 := X[i].0;
			L[i].0 := X[i].0;
		ELSIF temp.1 THEN
			code := 2;
			code.7 := X[i].1;
			L[i].1 := X[i].1;
		ELSIF temp.2 THEN
			code := 3;
			code.7 := X[i].2;
			L[i].2 := X[i].2;
		ELSIF temp.3 THEN
			CODE := 4;
			CODE.7 := X[i].3;
			L[i].3 := X[i].3;
		ELSIF temp.4 THEN
			CODE := 5;
			CODE.7 := X[i].4;
			L[i].4 := X[i].4;
		END_IF;
		TP := TRUE;
		CODE.4 := Line.0;
		CODE.5 := Line.1;
		CODE.6 := Line.2;

		(* check if release codes need to be killed *)
		IF NOT release AND CODE < 127 THEN
			CODE := 0;
			TP := FALSE;
		END_IF;
		EXIT;
	END_IF;
END_FOR;

(* increment scan line every cycle *)
line := (line + 1) AND 2#0000_0011;
temp := SHL(BYTE#1,line);
Y1 := temp.0;
Y2 := temp.1;
Y3 := temp.2;
Y4 := temp.3;




(* revision history
hm		10.6.2007	rev 1.0		
	original version 


hm		11.9.2007	rev 1.1		
	deleted unused variables k and old_code

hm		23.12.2007	rev 1.2
	added exit statement in for loop instead of i:=5

hm		26. oct. 2008	rev 1.3
	code optimized

*)
END_FUNCTION_BLOCK

(* POU MAX3, ST *)
FUNCTION MAX3 : REAL
VAR_INPUT
	in1 : REAL;
	in2 : REAL;
	in3 : REAL;
END_VAR
VAR
END_VAR

(*
version 1.0	1 jan 2007
programmer 	hugo
tested by		tobias

this function returns the highest of 3 real values

*)
IF in1 >= in2 AND in1 >= in3 THEN
	max3 := in1;
ELSIF in2 >= in1 AND in2 >= in3 THEN
	max3 := in2;
ELSE
	max3 := in3;
END_IF;
END_FUNCTION

(* POU MESSAGE_4R, ST *)
FUNCTION_BLOCK MESSAGE_4R
VAR_INPUT
	M0 : STRING(STRING_LENGTH);
	M1 : STRING(STRING_LENGTH);
	M2 : STRING(STRING_LENGTH);
	M3 : STRING(STRING_LENGTH);
	MM : INT := 3;
	ENQ : BOOL := TRUE;
	CLK : BOOL := TRUE;
	T1 : TIME := T#3s;
END_VAR
VAR_OUTPUT
	MX : STRING(STRING_LENGTH);
	MN : INT;
	TR : BOOL;
END_VAR
VAR
	timer : TON;
	edge: BOOL;
END_VAR

(*
version 1.1	27. oct. 2008
programmer 	hugo
tested by	tobias

this function generates a rotation meassage with up to 4 strings.
on each rising edge of EN the next message in line will be displayed.
when EN stays high longer then one cycle, the next message will be displayed automatically after the time T1 is elapsed.
the output MX is the generated message and CX is a counter 0..3 signaling the current message displayed.
the displayed messages are 0 .. MM.

*)
(* check for rising edge on EN *)
TR := FALSE;
IF ENQ THEN
	IF (NOT edge AND clk) OR timer.q THEN
			MN := INC1(MN, MM);
			TR := TRUE;
			timer(in := FALSE);
			CASE MN OF
				0 : MX := M0;
				1 : MX := M1;
				2 : MX := M2;
				3 : MX := M3;
			END_CASE;
	END_IF;
	edge := clk;
	timer( in := CLK, pt := T1);
ELSE
	MX := '';
	MN := 0;
END_IF;




(* revision history
hm	8. oct. 2008	rev 1.0
	original version

hm	27. oct. 2008	rev 1.1
	changed _INC to INC1

*)
END_FUNCTION_BLOCK

(* POU MESSAGE_8, ST *)
FUNCTION_BLOCK MESSAGE_8
VAR_INPUT
	IN1 : BOOL;
	IN2 : BOOL;
	IN3 : BOOL;
	IN4 : BOOL;
	IN5 : BOOL;
	IN6 : BOOL;
	IN7 : BOOL;
	IN8 : BOOL;
END_VAR
VAR_INPUT CONSTANT
	S1 : STRING(STRING_LENGTH);
	S2 : STRING(STRING_LENGTH);
	S3 : STRING(STRING_LENGTH);
	S4 : STRING(STRING_LENGTH);
	S5 : STRING(STRING_LENGTH);
	S6 : STRING(STRING_LENGTH);
	S7 : STRING(STRING_LENGTH);
	S8 : STRING(STRING_LENGTH);
END_VAR
VAR_OUTPUT
	M : STRING(STRING_LENGTH);
END_VAR
VAR
END_VAR

(*
version 1.1	29. mar. 2008
programmer 	hugo
tested by	tobias

this function generates one out of 4 messages specified by S1 .. S8.
the selected message will be presented at the output M.
In1 has higher priority then In2 which has higher priority then IN3 and in8 has the lowest priority.
*)
(* check if an alarm is present if yes set the output M otherwise clear M *)
IF in1 THEN
	M := S1;
ELSIF in2 THEN
	M := S2;
ELSIF in3 THEN
	M := S3;
ELSIF in4 THEN
	M := S4;
ELSIF in5 THEN
	M := S5;
ELSIF in6 THEN
	M := S6;
ELSIF in7 THEN
	M := S7;
ELSIF in8 THEN
	M := S8;
ELSE
	M := '';
END_IF;

(* revision history
hm	26.12.2007		rev 1.0
	original version

hm	29. mar. 2008	rev 1.1
	changed STRING to STRING(STRING_LENGTH)
*)
END_FUNCTION_BLOCK

(* POU METER_STAT, ST *)
FUNCTION_BLOCK METER_STAT
VAR_INPUT
	IN : REAL;
	DI : DATE;
	RST : BOOL;
END_VAR
VAR_OUTPUT RETAIN
	Last_Day : REAL;
	Current_Day : REAL;
	Last_Week : REAL;
	Current_Week : REAL;
	Last_Month : REAL;
	Current_Month : REAL;
	Last_Year : REAL;
	Current_Year : REAL;
END_VAR
VAR RETAIN
	Year_Start : REAL;
	Month_Start : REAL;
	Week_Start : REAL;
	Day_Start : REAL;
	last_run: DATE;
END_VAR

(*
	version 1.1	7. oct. 2008
	programmer 	oscat
	tested BY	oscat

METER_STAT runs statistics of a metered value, it calculates the current week, day, month and year consumption and stores the corresponding last day, week, month and year value.

*)
IF rst THEN
	Last_Day := 0;
	Current_Day := 0;
	Day_start := IN;
	Last_week := 0;
	Current_week := 0;
	Week_start := in;
	Last_month := 0;
	Current_month := 0;
	month_start := in;
	last_year := 0;
	current_year := 0;
	year_start := in;
ELSE
	Current_Day := IN - Day_Start;
	Current_Week := In - Week_Start;
	Current_Month := IN - Month_Start;
	Current_Year := IN - Year_Start;
END_IF;

IF YEAR_OF_DATE(DI) > YEAR_OF_DATE(last_run) THEN
	(* a new year has started *)
	last_year := current_year;
	current_year := 0;
	year_start := in;
	last_month := current_month;
	current_month := 0;
	month_start := in;
	last_day := current_day;
	current_day := 0;
	day_start := in;
ELSIF MONTH_OF_DATE(DI) > MONTH_OF_DATE(last_run) THEN
	(* a new month has started, january is alrerady done by year change *)
	last_month := current_month;
	current_month := 0;
	month_start := in;
	last_day := current_day;
	current_day := 0;
	day_start := in;
ELSIF day_of_year(di) > day_of_year(last_run) THEN
	(* day has chaged, first day of year and first day of month has already been taken care of *)
	last_day := current_day;
	current_day := 0;
	day_start := in;
END_IF;
IF DAY_OF_WEEK(DI) < DAY_OF_WEEK(last_run) THEN
	(* a new week has started *)
	last_week := current_week;
	current_week := 0;
	week_start := in;
END_IF;
last_run := di;

(* revision history
hm	16. sep. 2007	rev 1.0
	original version

hm	7. oct. 2008	rev 1.1
	changed function year_to_year_of_date
	changed function month to month_of_date
	changed function weekday to day_of_week

*)
END_FUNCTION_BLOCK

(* POU MID3, ST *)
FUNCTION MID3 : REAL
VAR_INPUT
	in1 : REAL;
	in2 : REAL;
	in3 : REAL;
END_VAR
VAR
END_VAR

(*
version 1.1	1 jan 2007
programmer 	hugo
tested by		tobias

returns the mid value of 3 real inputs.

*)
IF (in1 <= in2) AND (in1 >= in3) OR (in1 >= in2) AND (in1 <= in3) THEN
	mid3 := in1;
ELSIF (in2 <= in1) AND (in2 >= in3) OR (in2 >= in1) AND (in2 <= in3) THEN
	mid3 := in2;
ELSE
	mid3 := in3;
END_IF;

(*
hm	1.1.2007	rev 1.1
	rewrote the function for better performance

*)
END_FUNCTION

(* POU MIN3, ST *)
FUNCTION MIN3 : REAL
VAR_INPUT
	in1 : REAL;
	in2 : REAL;
	in3 : REAL;
END_VAR
VAR
END_VAR

(*
version 1.0	1 jan 2007
programmer 	hugo
tested by		tobias

this function returns the lowest of 3 real values

*)
IF in1 <= in2 AND in1 <= in3 THEN
	min3 := in1;
ELSIF in2 <= in1 AND in2 <= in3 THEN
	min3 := in2;
ELSE
	min3 := in3;
END_IF;
END_FUNCTION

(* POU MINUTE_OF_DT, ST *)
FUNCTION MINUTE_OF_DT : INT
VAR_INPUT
	XDT : DT;
END_VAR
VAR
END_VAR


(*
	version 1.0	6. jun. 2008
	programmer 	oscat
	tested BY	oscat

MINUTE_OF_DT returns the current minute (minute of the hour) of a DT variable

*)
MINUTE_OF_DT := DWORD_TO_INT(DT_TO_DWORD(XDT) MOD 3600)/60;


(* revision history
hm		6.9.2008	rev 1.0
	original version


*)
END_FUNCTION

(* POU MINUTE_TO_TIME, ST *)
FUNCTION MINUTE_TO_TIME : TIME
VAR_INPUT
	input : REAL;
END_VAR
VAR
END_VAR

(*
version 1.1	14 mar 2008
programmer 	hugo
tested by	tobias

converts an amount of minutes in real to time
execution time on wago 750-841 =  17us
*) 
minute_to_time := DWORD_TO_TIME(REAL_TO_DWORD(input * 60000));


(* revision history
hm		4. aug 2006	rev 1.0
	original version

hm		14. mar 2008	rev 1.1
	rounded the input after the last digit

*)
END_FUNCTION

(* POU MIRROR, ST *)
FUNCTION MIRROR : STRING(STRING_LENGTH)
VAR_INPUT
	str : STRING(STRING_LENGTH);
END_VAR
VAR
	pi : POINTER TO ARRAY[1..255] OF BYTE;
	po : POINTER TO BYTE;
	lx: INT;
	i: INT;
END_VAR

(*
version 1.1	29. mar. 2008
programmer 	hugo
tested by	tobias

this function reverses an input string.

*)
pi := ADR(str);
po := ADR(mirror);
lx := LEN(str);
FOR i := lx TO 1 BY - 1 DO
	po^ := pi^[i];
	po := po + 1;
END_FOR;
(* close output string *)
po^:= 0;


(* revision histroy
hm	4. feb. 2008	rev 1.0
	original release

hm	29. mar. 2008	rev 1.1
	changed STRING to STRING(STRING_LENGTH)
*)	
END_FUNCTION

(* POU MIX, ST *)
FUNCTION MIX : REAL
VAR_INPUT
	A, B : REAL;
	M : REAL;
END_VAR
VAR
END_VAR

(*
version 1.0	19 nov 2007
programmer 	hugo
tested by		tobias

MIX is an analog Mixer. The Output is (1-M)*A + M*B.

*)
MIX := (1-M)*A + M*B;

(* revision history
hm	19. Nov 2007		rev 1.0
	original version
*)
END_FUNCTION

(* POU MONTH_BEGIN, ST *)
FUNCTION MONTH_BEGIN : DATE
VAR_INPUT
	idate : DATE;
END_VAR
VAR
END_VAR

(*
version 1.0	15. jun. 2008
programmer 	hugo
tested by	oscat

returns the date for the first day of the current month in the current year.

*)
MONTH_BEGIN := DWORD_TO_DATE(DATE_TO_DWORD(idate) - INT_TO_DWORD(DAY_OF_MONTH(idate) - 1) * 86400);



(* revision history
hm	15. jun. 2008	rev 1.0
	original version	


*)
END_FUNCTION

(* POU MONTH_END, ST *)
FUNCTION MONTH_END : DATE
VAR_INPUT
	IDATE : DATE;
END_VAR
VAR
END_VAR

(*
version 1.1	7. oct. 2008
programmer 	hugo
tested by	oscat

returns the date for the last day of the current month in the current year.

*)
MONTH_END := DWORD_TO_DATE(DATE_TO_DWORD(SET_DATE(YEAR_OF_DATE(idate),MONTH_OF_DATE(idate)+1,1)) - 86400);



(* revision history
hm	15. jun. 2008	rev 1.0
	original version	

hm	7. oct. 2008	rev 1.1
	changed function year to year_of_date
	changed function month to month_of_date

*)
END_FUNCTION

(* POU MS_TO_BFT, ST *)
FUNCTION MS_TO_BFT : INT
VAR_INPUT
	MS : REAL;
END_VAR
VAR
END_VAR

(*
version 1.0	12. jun 2008
programmer 	hugo
tested by	oscdat

this function converts wind speed from M/s to beaufort
*)
MS_TO_BFT := REAL_TO_INT(EXPT(MS * 1.196172, 0.666667));


(* revision history
hm	12. 6. 2008		rev 1.0
	original version

*)
END_FUNCTION

(* POU MS_TO_KMH, ST *)
FUNCTION MS_TO_KMH : REAL
VAR_INPUT
	ms : REAL;
END_VAR
VAR
END_VAR

(*
version 1.0	4 Feb 2007
programmer 	hugo
tested by		tobias

this function converts velocities from Meters / Second to Kilometers / hour.

*)
MS_TO_KMH := ms * 3.6;
END_FUNCTION

(* POU MUL_ADD, ST *)
FUNCTION MUL_ADD : REAL
VAR_INPUT
	X : REAL;
	K : REAL;
	O : REAL;
END_VAR
VAR
END_VAR

(*
version 1.1	11 nov 2007
programmer 	hugo
tested by		tobias

this function multiplies an input X with K and adds Offset O to the result.

*)
MUL_ADD := X * K + O;

(* revision history
hm	28. feb 2007
	original version

hm	11.nov 2007		rev 1.1
	deleted preset values for K and O this makes no sense for a function

*)
END_FUNCTION

(* POU MULTI_IN, ST *)
FUNCTION MULTI_IN : REAL
VAR_INPUT
	in_1 : REAL;
	in_2 : REAL;
	in_3 : REAL;
	default : REAL;
	in_min : REAL;
	in_max : REAL;
	mode : BYTE;
END_VAR
VAR
	count: INT;
	F1: BOOL;
	F2: BOOL;
	F3: BOOL;
END_VAR

(*

version 1.2	14. oct. 2008
programmer 	oscat
tested by	oscat

multi_in is a signal conditioning function which can be configured in 8 different ways.
it is used to read multiple sensors for the same value and protect the user from broken sensors or invalid data from sensors.

multi_in can be configured in different ways:
	mode = 0 means the the avg of the 3 inputs is used, this mode is the default mode.
	mode = 1 means in_1 is used.
	mode = 2 means in_2 is used.
	mode = 3 means in_3 is used.
	mode = 4 means default is used.
	mode = 5 means the lowest of the 3 external temperatures is used.
	mode = 6 means the higest externnal temperature is used.
	mode = 7 means the midlle input is used, if there are only two working, the lowest input is used.
	mode > 7 ,eans output is 0 at all times.
	in any config mode, an input higher then in_max or lower then in_min is ignored to prevent values from broken sensors or wires.
	if all inputs are higher then in_max or lower then in_min, a default value (default) is used.
*)
F1 :=  in_1 > in_min AND in_1 < in_max;
F2 :=  in_2 > in_min AND in_2 < in_max;
F3 :=  in_3 > in_min AND in_3 < in_max;

CASE mode OF
0:	count := 0;
	IF F1 THEN
		count := count + 1;
		MULTI_IN := in_1;
	ELSE
		MULTI_IN := 0;
	END_IF;
	IF F2 THEN
		count := count + 1;
		MULTI_IN := MULTI_IN + in_2;
	END_IF;
	IF F3 THEN
		count := count + 1;
		MULTI_IN := MULTI_IN + in_3;
	END_IF;
	IF count = 0 THEN
		MULTI_IN := default;
	ELSE
		MULTI_IN := MULTI_IN / count;
	END_IF;

1:	IF F1 THEN MULTI_IN := in_1; ELSE MULTI_IN := default; END_IF;

2:	IF F2 THEN MULTI_IN := in_2; ELSE MULTI_IN := default; END_IF;

3:	IF F3 THEN MULTI_IN := in_3; ELSE MULTI_IN := default; END_IF;

4:	MULTI_IN := default;

5:	IF F1 THEN MULTI_IN := in_1; ELSE MULTI_IN := in_max; END_IF;
	IF F2 AND in_2 < MULTI_IN THEN MULTI_IN := in_2; END_IF;
	IF F3 AND in_3 < MULTI_IN THEN MULTI_IN := in_3; END_IF;
	IF MULTI_IN = in_max THEN MULTI_IN := default; END_IF;

6:	IF F1 THEN MULTI_IN := in_1; ELSE MULTI_IN := in_min; END_IF;
	IF F2 AND in_2 > MULTI_IN THEN MULTI_IN := in_2; END_IF;
	IF F3 AND in_3 > MULTI_IN THEN MULTI_IN := in_3; END_IF;
	IF MULTI_IN = in_min THEN MULTI_IN := default; END_IF;

7:	IF F1 AND F2 AND F3 THEN MULTI_IN := MID3(in_1, in_2, in_3);
	ELSIF F1 AND F2 THEN MULTI_IN := MIN(in_1, in_2);
	ELSIF F1 AND F3 THEN MULTI_IN := MIN(in_1, in_3);
	ELSIF F2 AND F3 THEN MULTI_IN := MIN(in_2, in_3);
	ELSIF F1 THEN MULTI_IN := in_1;
	ELSIF F2 THEN MULTI_IN := in_2;
	ELSIF F3 THEN MULTI_IN := in_3;
	ELSE MULTI_IN := default;
	END_IF;

END_CASE;

(*
hm 1.1.2007			rev 1.1
	changed midr to mid3 function

hm	14. 10. 2008	rev 1.2
	corrected an error for in_3 overrange detection
	improved performance


*)
END_FUNCTION

(* POU MUX_2, ST *)
FUNCTION MUX_2 : BOOL
VAR_INPUT
	D0: BOOL;
	D1: BOOL;
	A0: BOOL;
END_VAR
VAR
END_VAR

(*
	version 1.2	16. oct. 2008
	programmer 	hugo
	tested BY	oscat

	dual input multiplexer
	depending on the value of A0, D0 or D1 will be switched to the Output

	executioin TIME on wago 750-841 = 7us
*)
MUX_2 := SEL(A0, D0, D1);


(*
revision history:
hm	5.10.2006		rev 1.1
	changed to ST Langage for better portability.

hm	16. oct. 2008	rev 1.2
	improved performance

*)
END_FUNCTION

(* POU MUX_4, ST *)
FUNCTION MUX_4 : BOOL
VAR_INPUT
	D0: BOOL;
	D1: BOOL;
	D2: BOOL;
	D3: BOOL;
	A0: BOOL;
	A1: BOOL;
END_VAR
VAR
END_VAR

(*
version 1.2	16. oct. 2008
programmer 	hugo
tested BY	oscat

quad input multiplexer
depending on the value of A0 and A1, one of the 4 inputs will be switched to the Output


*)
IF A1 THEN
	MUX_4 := SEL(A0, D2, D3);
ELSE
	MUX_4 := SEL(A0, D0, D1);
END_IF;


(*
revision history:
hm 	5.10.2006		rev 1.1
	rewritten to ST for better portability

hm	16. oct. 2008	rev 1.2
	improved performance

*)
END_FUNCTION

(* POU MUX_R2, ST *)
FUNCTION MUX_R2 : REAL
VAR_INPUT
	IN0 : REAL;
	IN1 : REAL;
	A : BOOL;
END_VAR
VAR
END_VAR

(*
version 1.1	16. oct. 2008
programmer 	oscat
tested by	oscat

MUX_R2 is an analog Multiplexer.
one of 2 real inputs are selected and put through to out.
The Adress input A selects between 2 Real inputs IN0 and IN1, A=0 > In0, A=1 > in1.

*)
MUX_R2 := SEL(A, IN0, IN1);


(* revision history
hm	19. jan. 2007	rev 1.0
	original version

hm	16. oct. 2008	rev 1.1
	improved performance


*)
END_FUNCTION

(* POU MUX_R4, ST *)
FUNCTION MUX_R4 : REAL
VAR_INPUT
	IN0 : REAL;
	IN1 : REAL;
	IN2 : REAL;
	IN3 : REAL;
	A0 : BOOL;
	A1 : BOOL;
END_VAR
VAR
END_VAR

(*
version 1.1	16. oct. 2008
programmer 	oscat
tested by	oscat

MUX_R4 is an analog Multiplexer.
one of 4 real inputs are selected and put through to out.
The Adress input A0 and A1 selects between the 4 Real inputs IN0.. IN1.

*)
IF A1 THEN
	MUX_R4 := SEL(A0, IN2, IN3);
ELSE
	MUX_R4 := SEL(A0, IN0, IN1);
END_IF;



(* revision history
hm	19. jan 2007	rev 1.0
	original version

hm	16. oct. 2008	rev 1.1
	improved performance
*)
END_FUNCTION

(* POU NEGX, ST *)
FUNCTION NEGX : REAL
VAR_INPUT
	X : REAL;
END_VAR
VAR
END_VAR


(*
version 1.0	26. oct. 2008
programmer 	hugo
tested by	tobias

This function returns -X

*)
NEGX := -X;




(* revision history
hm	26. oct. 2008	rev 1.0
	original version


*)
END_FUNCTION

(* POU OFFSET2, ST *)
FUNCTION OFFSET2 : REAL
VAR_INPUT
	X : REAL;
	O1, O2, O3, O4 : BOOL;
	D : BOOL;
END_VAR
VAR_INPUT CONSTANT
	Offset_1 : REAL;
	Offset_2 : REAL;
	Offset_3 : REAL;
	Offset_4 : REAL;
	default : REAL;
END_VAR

(*
version 1.0	12 jan 2007
programmer 	oscat
tested by		tobias

The Function offset adds offsets to an analog signal depending on digital inputs.
one offset can be added at the same time, if more then one input is true, the one with the highest number (o1 .. o4) will be used.
The input D will select a default value instead of X for input.

*) 
IF D THEN OFFSET2 := default; ELSE OFFSET2 := X; END_IF;
IF O4 THEN OFFSET2 := OFFSET2 + offset_4;
ELSIF O3 THEN OFFSET2 := OFFSET2 + offset_3;
ELSIF O2 THEN OFFSET2 := OFFSET2 + offset_2;
ELSIF O1 THEN OFFSET2 := OFFSET2 + offset_1;
END_IF;
END_FUNCTION

(* POU OM_TO_F, ST *)
FUNCTION OM_TO_F : REAL
VAR_INPUT
	OM : REAL;
END_VAR
VAR
END_VAR

(*
version 1.1	18. oct. 2008
programmer 	hugo
tested by		tobias

this function converts Omega F to frequency
F = OM / (2*PI)
*)
OM_TO_F := OM / math.PI2;


(* revision history
hm	22. jan. 2007	rev 1.0
	original version

hm	18. oct. 2008	rev 1.1
	using math constants

*)
END_FUNCTION

(* POU OSCAT_VERSION, ST *)
FUNCTION OSCAT_VERSION : DWORD
VAR_INPUT
	IN : BOOL;
END_VAR
VAR
END_VAR


(*
version 1.1	16 dec 2007
programmer 	hugo
tested by	oscat

oscat_version returns the version number in dword format
132 is library version 1.32
if IN = true, the release date will be returned

*)
IF in THEN
	OSCAT_VERSION := DATE_TO_DWORD(D#2008-11-15);
ELSE
	OSCAT_VERSION := 302;
END_IF;

(* revision history
hm	6. oct 2006	rev 1.0
	original version

hm	16. dec 2007	rev 1.1
	added possibility to return date and version depending on IN.

*)
END_FUNCTION

(* POU OVERRIDE, ST *)
FUNCTION OVERRIDE : REAL
VAR_INPUT
	X1, X2, X3 : REAL;
	E1 : BOOL;
	E2 : BOOL;
	E3 : BOOL;
END_VAR
VAR
END_VAR

(*
version 1.0	4 nov 2007
programmer 	oscat
tested by	tobias

OVERRIDE deliveres the maximum absolute value of the 3 inputs X1, X2 and X3.
with the inputs E1, E2 and E3 each of the 3 inputs can be turned on or off.

*) 
IF E1 THEN OVERRIDE := X1; END_IF;
IF E2 AND ABS(x2) > ABS(OVERRIDE) THEN OVERRIDE := X2; END_IF;
IF E3 AND ABS(x3) > ABS(OVERRIDE) THEN OVERRIDE := X3; END_IF;

(* revision history
hm	4.11.2007		rev 1.0
	original version

*)
END_FUNCTION

(* POU PARITY, ST *)
FUNCTION PARITY : BOOL
VAR_INPUT
	in : DWORD;
END_VAR
VAR
END_VAR

(*
	version 1.3	18 feb 2008
	programmer 	hugo
	tested BY		hans

this function calculates the even parity of an input Dword
the output will be true if the amount of high bits are an odd number.

*)
WHILE in > 0 DO
	PARITY := PARITY XOR in.0 XOR in.1 XOR in.2 XOR in.3;
	in := SHR(in,4);
END_WHILE;

(* code before rev 1.2
WHILE in > 0 DO
	IF in.0 THEN cnt := cnt +1; END_IF;
	in := SHR(in,1);
END_WHILE;
IF (cnt MOD 2) = 1 THEN parity := TRUE; ELSE parity := FALSE; END_IF;
*)

(* revision history

rev 1.0 hm 1 sep 2006
	original version

rev 1.1 hm 10.9.2007
	changed algorithm to improve performance

rev 1.2	hm	8 dec 2007
	changed algorithm to improve performance

rev 1.3	hm	18 feb 2008
	changed algorithm to improve performance
*)
END_FUNCTION

(* POU PARSET, ST *)
FUNCTION_BLOCK PARSET
VAR_INPUT
	A0, A1 : BOOL;
END_VAR
VAR_INPUT CONSTANT
	X01, X02, X03, X04 : REAL;
	X11, X12, X13, X14 : REAL;
	X21, X22, X23, X24 : REAL;
	X31, X32, X33, X34 : REAL;
	TC : TIME;
END_VAR
VAR_OUTPUT
	P1, P2, P3, P4 : REAL;
END_VAR
VAR
	X : ARRAY[0..3,1..4] OF REAL;
	S1, S2, S3, S4 : REAL;
	tx, last : DWORD;
	start : BOOL;
	set : BYTE;
	init: BOOL;
END_VAR

(*
version 1.1	16. mar. 2008
programmer 	hugo
tested by		tobias

parset selects on of 4 parameter sets adressed by the inputs A0 and A1. if TC is specified, the change of the outputs
is ramped by the time tc
*)
(* read system_time *)
tx := T_PLC_MS();

(* init sequence *)
IF NOT init THEN
	set.0 := NOT A0;
	init := TRUE;
	X[0,1] := X01;
	X[0,2] := X02;
	X[0,3] := X03;
	X[0,4] := X04;
	X[1,1] := X11;
	X[1,2] := X12;
	X[1,3] := X13;
	X[1,4] := X14;
	X[2,1] := X21;
	X[2,2] := X22;
	X[2,3] := X23;
	X[2,4] := X24;
	X[3,1] := X31;
	X[3,2] := X32;
	X[3,3] := X33;
	X[3,4] := X34;
	P1 := X01;
	P2 := X02;
	P3 := X03;
	P4 := X04;
END_IF;

(* check for input change *)
IF (A0 XOR set.0) OR (A1 XOR set.1) THEN
	(* a new set is selected *)
	set.0 := A0;
	set.1 := A1;
	IF tc > t#0s THEN
		start := TRUE;
		last := tx;
		(* save the step speed for the output changes in S *)
		S1 := (X[set,1] - P1)/DWORD_TO_REAL(TIME_TO_DWORD(tc));
		S2 := (X[set,2] - P2)/DWORD_TO_REAL(TIME_TO_DWORD(tc));
		S3 := (X[set,3] - P3)/DWORD_TO_REAL(TIME_TO_DWORD(tc));
		S4 := (X[set,4] - P4)/DWORD_TO_REAL(TIME_TO_DWORD(tc));
	END_IF;
ELSIF start AND tx - last < TIME_TO_DWORD(tc) THEN
	(* ramp the outputs to the new value *)
	P1 := X[set,1] - S1 * DWORD_TO_REAL(TIME_TO_DWORD(Tc) - tx + last);
	P2 := X[set,2] - S2 * DWORD_TO_REAL(TIME_TO_DWORD(Tc) - tx + last);
	P3 := X[set,3] - S3 * DWORD_TO_REAL(TIME_TO_DWORD(Tc) - tx + last);
	P4 := X[set,4] - S4 * DWORD_TO_REAL(TIME_TO_DWORD(Tc) - tx + last);
ELSE
	(* make sure outputs match the correct set values *)
	start := FALSE;
	P1 := X[set,1];
	P2 := X[set,2];
	P3 := X[set,3];
	P4 := X[set,4];
END_IF;

(* revision history
hm	2.11.2007		rev 1.0
	original version

hm	16. mar. 2008	rev 1.1
	added type conversions to avoid warnings under codesys 3.0

*)
END_FUNCTION_BLOCK

(* POU PARSET2, ST *)
FUNCTION_BLOCK PARSET2
VAR_INPUT
	X : REAL;
END_VAR
VAR_INPUT CONSTANT
	X01, X02, X03, X04 : REAL;
	X11, X12, X13, X14 : REAL;
	X21, X22, X23, X24 : REAL;
	X31, X32, X33, X34 : REAL;
	L1, L2, L3 : REAL;
	TC : TIME;
END_VAR
VAR_OUTPUT
	P1,P2,P3,P4 : REAL;
END_VAR
VAR
	Pset : parset;
	init: BOOL;
END_VAR

(*
version 1.0	3 nov 2007
programmer 	hugo
tested by	tobias

parset2 selects on of 4 parameter sets depending on the value of X. if TC is specified, the change of the outputs
is ramped by the time TC
*)
(* init sequence *)
IF NOT init THEN
	init := TRUE;
	pset(TC:=TC, X01:=X01, X02:=X02, X03:=X03, X04:=X04, X11:=X11, X12:=X12, X13:=X13, X14:=X14, X21:=X21, X22:=X22, X23:=X23, X24:=X24, X31:=X31, X32:=X32, X33:=X33, X34:=X34);
END_IF;
IF ABS(X) < L1 THEN
	pset(A0 := FALSE, A1 := FALSE);
ELSIF ABS(X) < L2 THEN
	pset(A0 := TRUE, A1 := FALSE);
ELSIF ABS(x) < L3 THEN
	pset(A0 := FALSE, A1 := TRUE);
ELSE
	pset(A0 := TRUE, A1 := TRUE);
END_IF;
P1 := pset.P1;
P2 := pset.P2;
P3 := pset.P3;
P4 := pset.P4;

(* revision history
hm		3.11.2007		rev 1.0
	original version

*)
END_FUNCTION_BLOCK

(* POU PERIOD, ST *)
FUNCTION PERIOD : BOOL
VAR_INPUT
	d1 : DATE;
	dx : DATE;
	d2 : DATE;
END_VAR
VAR
	day1, day2, dayx : INT;
END_VAR

(*
version 1.3	22. mar. 2008
programmer 	hugo
tested by		tobias

PERIOD checks if a given date is between two dates (d1 and d2) d1 is the starting date and d2 the last date for the period.
the years of the dates are ignored, so the function period cheks for a time period within a year independet of the year.

*)
day1 := DAY_OF_YEAR(d1);
day2 := DAY_OF_YEAR(d2);
dayx := DAY_OF_YEAR(dx);
IF NOT LEAP_OF_DATE(dx) AND dayx > 58 THEN dayx := dayx + 1; END_IF;
IF NOT LEAP_OF_DATE(d1) AND day1 > 58 THEN day1 := day1 + 1; END_IF;
IF NOT LEAP_OF_DATE(d2) AND day2 > 58 THEN day2 := day2 + 1; END_IF;

IF day2 < day1 THEN
	(* the period spans over the new year *)
	PERIOD := dayx <= day2 OR dayx >= day1;
ELSE
	PERIOD := dayx >= day1 AND dayx <= day2;
END_IF;

(* code before rev 1.2
yx := year(dx);
p1 := date_add(d1,0,0,0,yx - year(d1));
p2 := date_add(d2,0,0,0,yx - year(d2));

IF p2 >= p1 THEN
	period := dx <= p2  AND dx >= p1;
ELSE
	period := dx <= p2 OR dx >= p1;
END_IF;
*)


(* revision history

hm		19. sep 2007	rev 1.0
	original version

hm		20. sep 2007	rev 1.1
	corrected a problem with leap year

hm		4. jan 2008		rev 1.2
	changed code for better performance

hm		22. mar. 2008	rev 1.3
	function would deliver wrong results when d1, d2 or dx are a leap_year

*)
END_FUNCTION

(* POU PERIOD2, ST *)
FUNCTION PERIOD2 : BOOL
VAR_INPUT
	DP : ARRAY[0..3,0..1] OF DATE;
	DX : DATE;
END_VAR
VAR
END_VAR

(*
version 1.0	27. apr. 2008
programmer 	hugo
tested by	tobias

PERIOD2 checks if DX is within one of 4 periods and sets the output true if so.

*)
PERIOD2 := 	(DX >= DP[0,0] AND DX <= DP[0,1]) OR
			(DX >= DP[1,0] AND DX <= DP[1,1]) OR
			(DX >= DP[2,0] AND DX <= DP[2,1]) OR
			(DX >= DP[3,0] AND DX <= DP[3,1]);


(* revision history

hm		27. apr 2008	rev 1.0
	original version


*) 
END_FUNCTION

(* POU PIN_CODE, ST *)
FUNCTION_BLOCK PIN_CODE
VAR_INPUT
	CB : BYTE;
	E : BOOL;
END_VAR
VAR_INPUT CONSTANT
	PIN : STRING(8);
END_VAR
VAR_OUTPUT
	TP : BOOL;
END_VAR
VAR
	POS: INT := 1;
END_VAR

(*
version 1.0	30. oct. 2008
programmer 	hugo
tested by	oscat

MATRIX_CODE scans the input of a key_pad (MATRIX) for a sequence of characters.

*)
tp := FALSE;
IF e THEN
	IF CB = CODE(pin, pos) THEN
		pos := pos + 1;
		IF pos > LEN(PIN) THEN
			(* proper code is detected *)
			TP := TRUE;
			pos := 1;
		END_IF;
	ELSE
		pos := 1;
	END_IF;
END_IF;


(* revision history
hm	30. oct. 2008	rev 1.0		
	original version 


*)
END_FUNCTION_BLOCK

(* POU POLYNOM_INT, ST *)
FUNCTION POLYNOM_INT : REAL
VAR_INPUT
	X : REAL;
	XY : ARRAY[1..5,0..1] OF REAL;
	Pts : INT;
END_VAR
VAR
	I, J : INT;
	stop: INT;
END_VAR

(*
	version 1.2	22 feb 2008
	programmer 	oscat
	tested BY		oscat

POLYNOM_INT calculates an output based on a Polynom interpolation of up to 5 coordinates given in an array
the indut coordinates have to start at the lowest array position and must be sorted ba ascending X values.

*)
(*make sure n is bound within the array size *)
pts := MIN(pts, 5);

(* this part is only to calculate the polynom parameters, which are then stores in the Y array
	the array values, it is not needed during runtime, unless the parameters will change during runtime
	the remaining code without this setup code can be used within a function to calculate specific functions
	the content of the arrays is then used as constant values within the function *)

FOR i := 1 TO pts DO
	stop := i + 1;
   	FOR j := pts TO stop BY -1 DO
   		XY[j,1] := (XY[j,1] - XY[j-1,1]) / (XY[j,0] - XY[j-i,0]);
	END_FOR;
END_FOR;


(* this part is the actual calculation *)
POLYNOM_INT := 0;
FOR i := pts TO 1 BY -1 DO
       POLYNOM_INT := POLYNOM_INT * (X - XY[i,0]) + XY[i,1];
END_FOR;


(* revision history
hm		8. okt 2007		rev 1.0
	original version

hm		17. dec 2007	rev 1.1
	init makes no sense for a function

hm		22. feb 2008	rev 1.2
	improved performance
*)
END_FUNCTION

(* POU PT_TO_F, ST *)
FUNCTION PT_TO_F : REAL
VAR_INPUT
	PT : TIME;
END_VAR
VAR
END_VAR

(*
version 1.0	4 aug 2006
programmer 	hugo
tested by		tobias

this function converts periode time to frequency
*)
PT_to_F := 1000/DWORD_TO_REAL(TIME_TO_DWORD(PT));
END_FUNCTION

(* POU PULSE_LENGTH, ST *)
FUNCTION_BLOCK PULSE_LENGTH
VAR_INPUT
	in : BOOL;
END_VAR
VAR_OUTPUT
	short : BOOL;
	middle : BOOL;
	long : BOOL;
END_VAR
VAR_INPUT CONSTANT
	T_short : TIME := t#100ms;
	T_long : TIME := t#1s;
END_VAR
VAR
	tx : TIME;
	tn: TIME;
	edge : BOOL;
END_VAR

(*
version 1.1	15 sep 2007
programmer 	oscat
tested by	oscat

Pulse_length indicates on 3 outputs if an input pulse had been shorter than T_short (short = True), longer than T_long (long = True) or between T_short and T_long (middle = True).

*)
(* read system time *)
tx := DWORD_TO_TIME(T_PLC_MS());

(* reset outputs, they should only be active 1 cycle *)
short := FALSE;
Middle := FALSE;
long := FALSE;

(* detect rising edge *)
IF in AND NOT edge THEN
	edge := TRUE;
	tn := tx;

(* detect for falling edge *)
ELSIF NOT in AND edge THEN
	edge := FALSE;
	tn := tx - tn;
	IF tn < t_short THEN
		short := TRUE;
	ELSIF tn > t_long THEN
		long := TRUE;
	ELSE
		Middle := TRUE;
	END_IF;

(* generate long pulse as soon as T_long is reached *)
ELSIF in AND tx - tn > t_long THEN
	long := TRUE;
END_IF;


(* revision history

hm	15. feb 2006	rev 1.0
	original version

hm	15 sep 2007		rev 1.1
	replaced Time() with T_PLC_MS for compatibility and performance reasons

*)
END_FUNCTION_BLOCK

(* POU PULSE_T, ST *)
FUNCTION_BLOCK PULSE_T
VAR_INPUT
	IN : BOOL;
	T1 : TIME;
	T2 : TIME;
	RST : BOOL;
END_VAR
VAR_OUTPUT
	Q : BOOL;
END_VAR
VAR
	init: BOOL;
	last: TIME;
	tx: TIME;
	edge: BOOL;
END_VAR


(*
version 1.0	15. jul. 2008
programmer 	hugo
tested by	oscat

PULSE_T generates a pulse of length T2 if the input pulse is shorter than T1.
if the input pulse is longer than T1, the output follows the input.
and rising edge on in will kill a possible output pulse and generate a new pulse instead.

*)
tx := DWORD_TO_TIME(T_PLC_MS());
IF NOT init THEN
	init := TRUE;
	last := tx;
ELSIF RST THEN
	(* asynchronous reset *)
	Q := FALSE;
ELSIF IN AND NOT edge AND NOT Q THEN
	(* a rising edge on in will reversre the output status, if new pulse is startet the start time is stored in last *)
	last := tx;
	Q := TRUE;
ELSIF NOT IN AND edge AND ((tx - last) > T1) THEN
	(* a falling edge on IN will clear the output if in was high for more then T1 *)
	Q := FALSE;
ELSIF (tx - last) >= T2 THEN
	(* timeout for long pulse if second click did not occur or in stays high *)
	Q := FALSE;
END_IF;

edge := IN;

(* revision histroy
hm	15. jul. 2008	rev 1.0
	original release


*)	
END_FUNCTION_BLOCK

(* POU PWM_PW, ST *)
FUNCTION_BLOCK PWM_PW
VAR_INPUT
	F : REAL;
	PW : TIME;
END_VAR
VAR_OUTPUT
	Q : BOOL;
END_VAR
VAR
	clk: CLK_PRG;
	pulse: TP_X;
END_VAR

(*
version 1.4	19. oct. 2008
programmer 	oscat
tested BY	oscat

this signal generator generates a square wave signal which is specified by the frequency and the pulse width.
*)
IF F > 0 THEN
	CLK(PT := REAL_TO_TIME(1000/F));
	Pulse(in := clk.Q, pt := pw);
	Q := pulse.Q;
END_IF;

(* revision history

hm	25. feb 2007	rev 1.1
	recoded in st for better performance and better portability

hm	27. nov 2007	rev 1.2
	avoid divide by 0 when F = 0

hm	9. dec 2007		rev 1.3
	corrected an error with F = 0

hm	19. oct. 2008	rev 1.4
	changed type tp_r to TP_x brecause of name change

*)
END_FUNCTION_BLOCK

(* POU R2_ABS, ST *)
FUNCTION R2_ABS : REAL2
VAR_INPUT
	X : REAL2;
END_VAR
VAR
END_VAR

(*
version 1.0	21. mar. 2008
programmer 	hugo
tested by		tobias

R2_abs returns the absulute value of a double precision real.

*)
IF X.RX >= 0 THEN
	R2_ABS.RX := X.RX;
	R2_ABS.R1 := X.R1;
ELSE
	R2_ABS.RX := ABS(X.RX);
	R2_ABS.R1 := -X.R1;
END_IF;


(* revision history
hm	21. mar. 2008	rev 1.0
	original version

*)
END_FUNCTION

(* POU R2_ADD2, ST *)
FUNCTION R2_ADD2 : REAL2
VAR_INPUT
	X : Real2;
	Y : REAL2;
END_VAR
VAR
END_VAR

(*
version 1.0	20. mar. 2008
programmer 	hugo
tested by		tobias

R2_add2 adds a double precision real to a double precision real which extends the accuracy of a real to twice as many digits

*)
R2_ADD2.R1 := X.R1 + Y.R1;
R2_ADD2.RX := X.RX + Y.RX;


(* revision history
hm		20.3.2008	rev 1.0
	original version

*)
END_FUNCTION

(* POU R2_MUL, ST *)
FUNCTION R2_MUL : REAL2
VAR_INPUT
	X : REAL2;
	Y : REAL;
END_VAR
VAR
END_VAR

(*
version 1.0	20. mar. 2008
programmer 	hugo
tested by		tobias

R2_mul multiplies a real with a double real which extends the accuracy of a real to twice as many digits

*)
R2_MUL.RX := X.RX * Y;
R2_MUL.R1 := X.R1 * Y;


(* revision history
hm		20.3.2008	rev 1.0
	original version

*)
END_FUNCTION

(* POU RANGE_TO_BYTE, ST *)
FUNCTION RANGE_TO_BYTE : BYTE
VAR_INPUT
	X : REAL;
	low : REAL;
	high : REAL;
END_VAR
VAR
END_VAR

(*
version 1.0	9. jan 2008
programmer 	hugo
tested by		tobias

Range_to_byte converts a real value between low and high into a byte

*)
Range_to_Byte := INT_TO_BYTE(TRUNC((LIMIT(low,X,high)-low) * 255.0 / (high - low)));


(* revision history
hm	9. jan 2008		rev 1.0
	original version

*)
END_FUNCTION

(* POU RANGE_TO_WORD, ST *)
FUNCTION RANGE_TO_WORD : WORD
VAR_INPUT
	X : REAL;
	low : REAL;
	high : REAL;
END_VAR
VAR
END_VAR

(*
version 1.0	9. jan 2008
programmer 	hugo
tested by		tobias

Range_to_word converts a real value between low and high into a byte

*)
Range_to_Word := DINT_TO_WORD(TRUNC((LIMIT(low,X,high)-low) * 65535.0 / (high - low)));


(* revision history
hm	9. jan 2008		rev 1.0
	original version

*)
END_FUNCTION

(* POU RDMDW, ST *)
FUNCTION RDMDW : DWORD
VAR_INPUT
	last : DWORD;
END_VAR
VAR
	RX: REAL;
	M: REAL;
END_VAR




(*
version 1.2	18. oct. 2008
programmer 	hugo
tested by		tobias

this function calculates a DWORD pseudo random number.

*)
M := BIT_COUNT(last);
RX := RDM(FRACT(M * math.PI));
RDMDW := SHL(REAL_TO_DWORD(rx*65535),16);
RX := RDM(FRACT(M * math.E));
RDMDW := RDMDW OR (REAL_TO_DWORD(rx*65535) AND 16#0000FFFF);



(* revision history
hm		14. mar 2008		rev 1.0
	original version

hm		18. may. 2008		rev 1.1
	changed constant E to E1

hm		18. oct. 2008		rev 1.2
	using math constants

*)
END_FUNCTION

(* POU REAL_TO_DW, ST *)
FUNCTION REAL_TO_DW : DWORD
VAR_INPUT
	X : REAL;
END_VAR
VAR
	pt : POINTER TO DWORD;
END_VAR

(*
version 1.0	18. apr. 2008
programmer 	hugo
tested by		tobias

this function converts a 32 Bit Real to a dword in a bitwise manner.
*)
pt := ADR(X);
REAL_TO_DW := pt^;

(* revision history
hm	18. apr. 2008
	original version

*)
END_FUNCTION

(* POU REAL_TO_STRF, ST *)
FUNCTION REAL_TO_STRF : STRING(20)
VAR_INPUT
	IN : REAL;
	N : INT;
END_VAR
VAR
	O: REAL;
END_VAR

(*
version 1.6	4. apr. 2008
programmer 	hugo
tested by	tobias

Real_to_strF converts a Real to a fixed length String.
the string will be filles with zeroes to achieve the fixed length after the dot.


*)
N := LIMIT(0,N,20);
(* round the input to N digits and convert to string *)
O := in * EXP10(N);
REAL_TO_STRF := DINT_TO_STRING(REAL_TO_DINT(O));
IF LEN(REAL_TO_STRF) < N THEN REAL_TO_STRF := FIX(REAL_TO_STRF, N+1, 48, 1); END_IF;
IF N > 0 THEN REAL_TO_STRF := INSERT(REAL_TO_STRF,'.',LEN(REAL_TO_STRF)-N); END_IF;


(* code used for rev 1.2
(* read pointer to output *)
p1 := ADR(REAL_TO_STRF);
p2 := p1;

(* multiply in with 10^N and truncate *)
FOR I := 1 TO N DO
	temp := temp * 10;
END_FOR;
temp := TRUNC(in * temp + 0.5);
(* multiply temp with in to shift n digits to the left *)
REAL_TO_STRF := DWORD_TO_STRING(temp);
(* now take care of the dot at length - Nth position *)
L := LEN(REAL_TO_STRF);
(* we need to add zero's at the end of the string if there are less then N + 1 zeroes *)
(* this for loop is to align the pointer p1 to the end of the string *)
FOR i := 1 TO L DO p1 := p1 + 1; END_FOR;
FOR i := L TO N DO
	p1^ := 48;
	p1 := p1 + 1;
END_FOR;
(* now we create the space for the dot *)
p2 := p1 - 1;
FOR i := 1 TO N DO
	p1^ := p2^;
	p1 := p1 - 1;
	p2 := p2 - 1;
END_FOR;
(* now we add the dot if N > 0 *)
IF N > 0 THEN
	p1^ := 46;
	(* the string needs to be closed with a 0 at the end *)
	FOR i := 1 TO N + 1 DO p1 := p1 + 1; END_FOR;
	p1^ := 0;
END_IF;
*)

(* code before rev 1.2
dw1 := TRUNC(ABS(in));
dw2 := TRUNC(fract(ABS(in))*exp10(N)+0.5);
IF in < 0 THEN
	s1 := CONCAT('-', DWORD_TO_STRING(dw1));
ELSE
	s1 := DWORD_TO_STRING(dw1);
END_IF;
IF N > 0 THEN s1 := CONCAT(s1, '.'); END_IF;
s2 := DWORD_To_STRF(dw2,N);
Real_To_StrF := CONCAT(s1, s2);
*)

(* revision history
hm		26 jan 2007	rev 1.0
	original version

hm	20. nov. 2007	rev 1.1
	when N=0 ther will be no dot at the end of the string.

hm	15. dec. 2007	rev 1.2
	changed code for better performance

hm	4. mar. 2008	rev 1.3
	result is now rounded instead of trunc

hm	20. mar. 2008	rev 1.4
	changed trunc to real_to_dint because trunc was generating wrong values on wago 842

hm	29. mar. 2008	rev 1.5
	changed STRING to STRING(20)

hm	4. apr. 2008	rev 1.6
	added variable O to avoid an error uner CoDeSys SP PLCWinNT V2.4
*)
END_FUNCTION

(* POU REFRACTION, ST *)
FUNCTION REFRACTION : REAL
VAR_INPUT
	ELEV : REAL;
END_VAR
VAR
	tmp: REAL;
END_VAR


(*
version 1.0	14. jul. 2008
programmer 	hugo
tested by	oscat

REFRACTION calculates the atmospheric refraction in degrees.
the input nangle goes from 0 at the hirizon to 90 at midday.

